gfCNCPoint1[25204] = {X 212.6141, Y 102.4000, Z -2.1667, A 0.000, B 0.000, C 0.000 }
gfCNCPoint1[25205] = {X 194.9870, Y 102.4000, Z -2.1667, A 0.000, B 0.000, C 0.000 }
gfCNCPoint1[25206] = {X 194.0079, Y 102.2897, Z -2.1667, A 0.000, B 0.000, C 0.000 }
gfCNCPoint1[25207] = {X 193.0779, Y 101.9643, Z -2.1667, A 0.000, B 0.000, C 0.000 }
gfCNCPoint1[25208] = {X 192.2436, Y 101.4401, Z -2.1667, A 0.000, B 0.000, C 0.000 }
gfCNCPoint1[25209] = {X 191.5469, Y 100.7434, Z -2.1667, A 0.000, B 0.000, C 0.000 }
gfCNCPoint1[25210] = {X 191.0227, Y 99.9091, Z -2.1667, A 0.000, B 0.000, C 0.000 }
gfCNCPoint1[25211] = {X 190.6973, Y 98.9791, Z -2.1667, A 0.000, B 0.000, C 0.000 }
gfCNCPoint1[25212] = {X 190.5870, Y 98.0000, Z -2.1667, A 0.000, B 0.000, C 0.000 }
gfCNCPoint1[25213] = {X 190.5870, Y 97.0659, Z -2.1667, A 0.000, B 0.000, C 0.000 }
gfCNCPoint1[25214] = {X 190.6897, Y 96.1207, Z -2.1667, A 0.000, B 0.000, C 0.000 }
gfCNCPoint1[25215] = {X 190.9931, Y 95.2196, Z -2.1667, A 0.000, B 0.000, C 0.000 }
gfCNCPoint1[25216] = {X 191.4830, Y 94.4047, Z -2.1667, A 0.000, B 0.000, C 0.000 }
gfCNCPoint1[25217] = {X 188.5295, Y 91.1802, Z -2.1667, A 0.000, B 0.000, C 0.000 }
gfCNCPoint1[25218] = {X 150.1254, Y 91.1802, Z -2.1667, A 0.000, B 0.000, C 0.000 }
gfCNCPoint1[25219] = {X 147.2491, Y 94.3668, Z -2.1667, A 0.000, B 0.000, C 0.000 }
gfCNCPoint1[25220] = {X 147.7550, Y 95.1910, Z -2.1667, A 0.000, B 0.000, C 0.000 }
gfCNCPoint1[25221] = {X 148.0700, Y 96.1053, Z -2.1667, A 0.000, B 0.000, C 0.000 }
gfCNCPoint1[25222] = {X 148.1791, Y 97.0661, Z -2.1667, A 0.000, B 0.000, C 0.000 }
gfCNCPoint1[25223] = {X 148.1791, Y 98.0000, Z -2.1667, A 0.000, B 0.000, C 0.000 }
gfCNCPoint1[25224] = {X 148.0688, Y 98.9791, Z -2.1667, A 0.000, B 0.000, C 0.000 }
gfCNCPoint1[25225] = {X 147.7434, Y 99.9091, Z -2.1667, A 0.000, B 0.000, C 0.000 }
gfCNCPoint1[25226] = {X 147.2192, Y 100.7434, Z -2.1667, A 0.000, B 0.000, C 0.000 }
gfCNCPoint1[25227] = {X 146.5225, Y 101.4401, Z -2.1667, A 0.000, B 0.000, C 0.000 }
gfCNCPoint1[25228] = {X 145.6882, Y 101.9643, Z -2.1667, A 0.000, B 0.000, C 0.000 }
gfCNCPoint1[25229] = {X 144.7582, Y 102.2897, Z -2.1667, A 0.000, B 0.000, C 0.000 }
gfCNCPoint1[25230] = {X 143.7791, Y 102.4000, Z -2.1667, A 0.000, B 0.000, C 0.000 }
gfCNCPoint1[25231] = {X 125.0000, Y 102.4000, Z -2.1667, A 0.000, B 0.000, C 0.000 }
gfCNCPoint1[25232] = {X 124.0209, Y 102.2897, Z -2.1667, A 0.000, B 0.000, C 0.000 }
gfCNCPoint1[25233] = {X 123.0909, Y 101.9643, Z -2.1667, A 0.000, B 0.000, C 0.000 }
gfCNCPoint1[25234] = {X 122.2566, Y 101.4401, Z -2.1667, A 0.000, B 0.000, C 0.000 }
gfCNCPoint1[25235] = {X 121.5599, Y 100.7434, Z -2.1667, A 0.000, B 0.000, C 0.000 }
gfCNCPoint1[25236] = {X 121.0357, Y 99.9091, Z -2.1667, A 0.000, B 0.000, C 0.000 }
gfCNCPoint1[25237] = {X 120.7103, Y 98.9791, Z -2.1667, A 0.000, B 0.000, C 0.000 }
gfCNCPoint1[25238] = {X 120.6000, Y 98.0000, Z -2.1667, A 0.000, B 0.000, C 0.000 }
gfCNCPoint1[25239] = {X 120.6000, Y 97.0659, Z -2.1667, A 0.000, B 0.000, C 0.000 }
gfCNCPoint1[25240] = {X 120.7047, Y 96.1117, Z -2.1667, A 0.000, B 0.000, C 0.000 }
gfCNCPoint1[25241] = {X 121.0139, Y 95.2029, Z -2.1667, A 0.000, B 0.000, C 0.000 }
gfCNCPoint1[25242] = {X 121.5128, Y 94.3828, Z -2.1667, A 0.000, B 0.000, C 0.000 }
gfCNCPoint1[25243] = {X 122.1777, Y 93.6904, Z -2.1667, A 0.000, B 0.000, C 0.000 }
gfCNCPoint1[25244] = {X 122.9769, Y 93.1586, Z -2.1667, A 0.000, B 0.000, C 0.000 }
gfCNCPoint1[25245] = {X 123.8724, Y 92.8129, Z -2.1667, A 0.000, B 0.000, C 0.000 }
gfCNCPoint1[25246] = {X 124.8216, Y 92.6696, Z -2.1667, A 0.000, B 0.000, C 0.000 }
gfCNCPoint1[25247] = {X 124.8681, Y 92.6535, Z -2.1667, A 0.000, B 0.000, C 0.000 }
gfCNCPoint1[25248] = {X 124.9163, Y 92.6433, Z -2.1667, A 0.000, B 0.000, C 0.000 }
gfCNCPoint1[25249] = {X 125.4404, Y 92.5656, Z -2.1667, A 0.000, B 0.000, C 0.000 }
gfCNCPoint1[25250] = {X 126.2564, Y 92.4277, Z -2.1667, A 0.000, B 0.000, C 0.000 }
gfCNCPoint1[25251] = {X 127.0615, Y 92.2363, Z -2.1667, A 0.000, B 0.000, C 0.000 }
gfCNCPoint1[25252] = {X 128.2733, Y 91.0927, Z -2.1667, A 0.000, B 0.000, C 0.000 }
gfCNCPoint1[25253] = {X 129.4217, Y 89.8854, Z -2.1667, A 0.000, B 0.000, C 0.000 }
gfCNCPoint1[25254] = {X 133.5081, Y 85.3901, Z -2.1667, A 0.000, B 0.000, C 0.000 }
gfCNCPoint1[25255] = {X 155.5332, Y 61.2114, Z -2.1667, A 0.000, B 0.000, C 0.000 }
gfCNCPoint1[25256] = {X 155.1842, Y 60.4951, Z -2.1667, A 0.000, B 0.000, C 0.000 }
gfCNCPoint1[25257] = {X 154.9701, Y 59.7276, Z -2.1667, A 0.000, B 0.000, C 0.000 }
gfCNCPoint1[25258] = {X 154.8980, Y 58.9340, Z -2.1667, A 0.000, B 0.000, C 0.000 }
gfCNCPoint1[25259] = {X 154.8980, Y 58.0000, Z -2.1667, A 0.000, B 0.000, C 0.000 }
gfCNCPoint1[25260] = {X 155.0083, Y 57.0209, Z -2.1667, A 0.000, B 0.000, C 0.000 }
gfCNCPoint1[25261] = {X 155.3337, Y 56.0909, Z -2.1667, A 0.000, B 0.000, C 0.000 }
gfCNCPoint1[25262] = {X 155.8579, Y 55.2566, Z -2.1667, A 0.000, B 0.000, C 0.000 }
gfCNCPoint1[25263] = {X 156.5546, Y 54.5599, Z -2.1667, A 0.000, B 0.000, C 0.000 }
gfCNCPoint1[25264] = {X 157.3889, Y 54.0357, Z -2.1667, A 0.000, B 0.000, C 0.000 }
gfCNCPoint1[25265] = {X 158.3189, Y 53.7103, Z -2.1667, A 0.000, B 0.000, C 0.000 }
gfCNCPoint1[25266] = {X 159.2980, Y 53.6000, Z -2.1667, A 0.000, B 0.000, C 0.000 }
gfCNCPoint1[25267] = {X 178.5335, Y 53.6000, Z -2.1667, A 0.000, B 0.000, C 0.000 }
gfCNCPoint1[25268] = {X 179.5126, Y 53.7103, Z -2.1667, A 0.000, B 0.000, C 0.000 }
gfCNCPoint1[25269] = {X 180.4426, Y 54.0357, Z -2.1667, A 0.000, B 0.000, C 0.000 }
gfCNCPoint1[25270] = {X 181.2769, Y 54.5599, Z -2.1667, A 0.000, B 0.000, C 0.000 }
gfCNCPoint1[25271] = {X 181.9736, Y 55.2566, Z -2.1667, A 0.000, B 0.000, C 0.000 }
gfCNCPoint1[25272] = {X 182.4978, Y 56.0909, Z -2.1667, A 0.000, B 0.000, C 0.000 }
gfCNCPoint1[25273] = {X 182.8232, Y 57.0209, Z -2.1667, A 0.000, B 0.000, C 0.000 }
gfCNCPoint1[25274] = {X 182.9335, Y 58.0000, Z -2.1667, A 0.000, B 0.000, C 0.000 }
gfCNCPoint1[25275] = {X 182.9334, Y 58.9704, Z -2.1667, A 0.000, B 0.000, C 0.000 }
gfCNCPoint1[25276] = {X 182.8587, Y 59.7421, Z -2.1667, A 0.000, B 0.000, C 0.000 }
gfCNCPoint1[25277] = {X 182.6497, Y 60.4886, Z -2.1667, A 0.000, B 0.000, C 0.000 }
gfCNCPoint1[25278] = {X 182.3130, Y 61.1869, Z -2.1667, A 0.000, B 0.000, C 0.000 }
gfCNCPoint1[25279] = {X 209.5365, Y 90.8998, Z -2.1667, A 0.000, B 0.000, C 0.000 }
gfCNCPoint1[25280] = {X 210.1906, Y 91.5634, Z -2.1667, A 0.000, B 0.000, C 0.000 }
gfCNCPoint1[25281] = {X 210.8912, Y 92.1776, Z -2.1667, A 0.000, B 0.000, C 0.000 }
gfCNCPoint1[25282] = {X 211.1525, Y 92.3423, Z -2.1667, A 0.000, B 0.000, C 0.000 }
gfCNCPoint1[25283] = {X 211.4457, Y 92.4397, Z -2.1667, A 0.000, B 0.000, C 0.000 }
gfCNCPoint1[25284] = {X 212.1215, Y 92.5841, Z -2.1667, A 0.000, B 0.000, C 0.000 }
gfCNCPoint1[25285] = {X 213.4014, Y 92.7454, Z -2.1667, A 0.000, B 0.000, C 0.000 }
gfCNCPoint1[25286] = {X 214.4545, Y 92.6566, Z -2.1667, A 0.000, B 0.000, C 0.000 }
gfCNCPoint1[25287] = {X 215.5097, Y 92.5965, Z -2.1667, A 0.000, B 0.000, C 0.000 }
gfCNCPoint1[25288] = {X 216.1638, Y 92.5242, Z -2.1667, A 0.000, B 0.000, C 0.000 }
gfCNCPoint1[25289] = {X 216.7936, Y 92.3335, Z -2.1667, A 0.000, B 0.000, C 0.000 }
gfCNCPoint1[25290] = {X 217.3779, Y 92.0307, Z -2.1667, A 0.000, B 0.000, C 0.000 }
gfCNCPoint1[25291] = {X 222.9188, Y 88.4548, Z -2.1667, A 0.000, B 0.000, C 0.000 }
gfCNCPoint1[25292] = {X 245.6538, Y 73.9166, Z -2.1667, A 0.000, B 0.000, C 0.000 }
gfCNCPoint1[25293] = {X 221.6008, Y 64.4770, Z -2.1667, A 0.000, B 0.000, C 0.000 }
gfCNCPoint1[25294] = {X 219.8423, Y 63.8884, Z -2.1667, A 0.000, B 0.000, C 0.000 }
gfCNCPoint1[25295] = {X 218.0280, Y 63.5049, Z -2.1667, A 0.000, B 0.000, C 0.000 }
gfCNCPoint1[25296] = {X 216.1817, Y 63.3315, Z -2.1667, A 0.000, B 0.000, C 0.000 }
gfCNCPoint1[25297] = {X 215.2275, Y 63.1935, Z -2.1667, A 0.000, B 0.000, C 0.000 }
gfCNCPoint1[25298] = {X 214.3263, Y 62.8509, Z -2.1667, A 0.000, B 0.000, C 0.000 }
gfCNCPoint1[25299] = {X 213.5213, Y 62.3203, Z -2.1667, A 0.000, B 0.000, C 0.000 }
gfCNCPoint1[25300] = {X 212.8512, Y 61.6271, Z -2.1667, A 0.000, B 0.000, C 0.000 }
gfCNCPoint1[25301] = {X 212.3482, Y 60.8047, Z -2.1667, A 0.000, B 0.000, C 0.000 }
gfCNCPoint1[25302] = {X 212.0364, Y 59.8924, Z -2.1667, A 0.000, B 0.000, C 0.000 }
gfCNCPoint1[25303] = {X 211.9308, Y 58.9340, Z -2.1667, A 0.000, B 0.000, C 0.000 }
gfCNCPoint1[25304] = {X 211.9308, Y 58.0000, Z -2.1667, A 0.000, B 0.000, C 0.000 }
gfCNCPoint1[25305] = {X 212.0411, Y 57.0209, Z -2.1667, A 0.000, B 0.000, C 0.000 }
gfCNCPoint1[25306] = {X 212.3665, Y 56.0909, Z -2.1667, A 0.000, B 0.000, C 0.000 }
gfCNCPoint1[25307] = {X 212.8907, Y 55.2566, Z -2.1667, A 0.000, B 0.000, C 0.000 }
gfCNCPoint1[25308] = {X 213.5875, Y 54.5599, Z -2.1667, A 0.000, B 0.000, C 0.000 }
gfCNCPoint1[25309] = {X 214.4217, Y 54.0357, Z -2.1667, A 0.000, B 0.000, C 0.000 }
gfCNCPoint1[25310] = {X 215.3517, Y 53.7103, Z -2.1667, A 0.000, B 0.000, C 0.000 }
gfCNCPoint1[25311] = {X 216.3308, Y 53.6000, Z -2.1667, A 0.000, B 0.000, C 0.000 }
gfCNCPoint1[25312] = {X 237.2617, Y 53.6000, Z -2.1667, A 0.000, B 0.000, C 0.000 }
gfCNCPoint1[25313] = {X 238.2408, Y 53.7103, Z -2.1667, A 0.000, B 0.000, C 0.000 }
gfCNCPoint1[25314] = {X 239.1708, Y 54.0357, Z -2.1667, A 0.000, B 0.000, C 0.000 }
gfCNCPoint1[25315] = {X 240.0050, Y 54.5599, Z -2.1667, A 0.000, B 0.000, C 0.000 }
gfCNCPoint1[25316] = {X 240.7017, Y 55.2566, Z -2.1667, A 0.000, B 0.000, C 0.000 }
gfCNCPoint1[25317] = {X 241.2260, Y 56.0909, Z -2.1667, A 0.000, B 0.000, C 0.000 }
gfCNCPoint1[25318] = {X 241.5514, Y 57.0209, Z -2.1667, A 0.000, B 0.000, C 0.000 }
gfCNCPoint1[25319] = {X 241.6617, Y 58.0000, Z -2.1667, A 0.000, B 0.000, C 0.000 }
gfCNCPoint1[25320] = {X 241.6617, Y 58.1782, Z -2.1667, A 0.000, B 0.000, C 0.000 }
gfCNCPoint1[25321] = {X 247.5187, Y 60.4616, Z -2.1667, A 0.000, B 0.000, C 0.000 }
gfCNCPoint1[25322] = {X 275.5538, Y 71.5851, Z -2.1667, A 0.000, B 0.000, C 0.000 }
gfCNCPoint1[25323] = {X 275.5530, Y 63.2813, Z -2.1667, A 0.000, B 0.000, C 0.000 }
gfCNCPoint1[25324] = {X 274.6937, Y 63.0561, Z -2.1667, A 0.000, B 0.000, C 0.000 }
gfCNCPoint1[25325] = {X 273.8971, Y 62.6630, Z -2.1667, A 0.000, B 0.000, C 0.000 }
gfCNCPoint1[25326] = {X 273.1956, Y 62.1178, Z -2.1667, A 0.000, B 0.000, C 0.000 }
gfCNCPoint1[25327] = {X 272.6180, Y 61.4429, Z -2.1667, A 0.000, B 0.000, C 0.000 }
gfCNCPoint1[25328] = {X 272.1877, Y 60.6657, Z -2.1667, A 0.000, B 0.000, C 0.000 }
gfCNCPoint1[25329] = {X 271.9224, Y 59.8179, Z -2.1667, A 0.000, B 0.000, C 0.000 }
gfCNCPoint1[25330] = {X 271.8327, Y 58.9340, Z -2.1667, A 0.000, B 0.000, C 0.000 }
gfCNCPoint1[25331] = {X 271.8327, Y 58.0000, Z -2.1667, A 0.000, B 0.000, C 0.000 }
gfCNCPoint1[25332] = {X 271.9430, Y 57.0209, Z -2.1667, A 0.000, B 0.000, C 0.000 }
gfCNCPoint1[25333] = {X 272.2684, Y 56.0909, Z -2.1667, A 0.000, B 0.000, C 0.000 }
gfCNCPoint1[25334] = {X 272.7926, Y 55.2566, Z -2.1667, A 0.000, B 0.000, C 0.000 }
gfCNCPoint1[25335] = {X 273.4893, Y 54.5599, Z -2.1667, A 0.000, B 0.000, C 0.000 }
gfCNCPoint1[25336] = {X 274.3236, Y 54.0357, Z -2.1667, A 0.000, B 0.000, C 0.000 }
gfCNCPoint1[25337] = {X 275.2536, Y 53.7103, Z -2.1667, A 0.000, B 0.000, C 0.000 }
gfCNCPoint1[25338] = {X 276.2327, Y 53.6000, Z -2.1667, A 0.000, B 0.000, C 0.000 }
gfCNCPoint1[25339] = {X 292.7731, Y 53.6000, Z -2.1667, A 0.000, B 0.000, C 0.000 }
gfCNCPoint1[25340] = {X 293.7522, Y 53.7103, Z -2.1667, A 0.000, B 0.000, C 0.000 }
gfCNCPoint1[25341] = {X 294.6822, Y 54.0357, Z -2.1667, A 0.000, B 0.000, C 0.000 }
gfCNCPoint1[25342] = {X 295.5164, Y 54.5599, Z -2.1667, A 0.000, B 0.000, C 0.000 }
gfCNCPoint1[25343] = {X 296.2131, Y 55.2566, Z -2.1667, A 0.000, B 0.000, C 0.000 }
gfCNCPoint1[25344] = {X 296.7373, Y 56.0909, Z -2.1667, A 0.000, B 0.000, C 0.000 }
gfCNCPoint1[25345] = {X 297.0628, Y 57.0209, Z -2.1667, A 0.000, B 0.000, C 0.000 }
gfCNCPoint1[25346] = {X 297.1731, Y 58.0000, Z -2.1667, A 0.000, B 0.000, C 0.000 }
gfCNCPoint1[25347] = {X 297.1731, Y 58.9355, Z -2.1667, A 0.000, B 0.000, C 0.000 }
gfCNCPoint1[25348] = {X 297.0808, Y 59.8184, Z -2.1667, A 0.000, B 0.000, C 0.000 }
gfCNCPoint1[25349] = {X 296.8139, Y 60.6650, Z -2.1667, A 0.000, B 0.000, C 0.000 }
gfCNCPoint1[25350] = {X 296.3831, Y 61.4411, Z -2.1667, A 0.000, B 0.000, C 0.000 }
gfCNCPoint1[25351] = {X 295.8058, Y 62.1154, Z -2.1667, A 0.000, B 0.000, C 0.000 }
gfCNCPoint1[25352] = {X 295.1053, Y 62.6607, Z -2.1667, A 0.000, B 0.000, C 0.000 }
gfCNCPoint1[25353] = {X 294.3099, Y 63.0548, Z -2.1667, A 0.000, B 0.000, C 0.000 }
gfCNCPoint1[25354] = {X 293.4518, Y 63.2820, Z -2.1667, A 0.000, B 0.000, C 0.000 }
gfCNCPoint1[25355] = {X 293.4518, Y 92.7117, Z -2.1667, A 0.000, B 0.000, C 0.000 }
gfCNCPoint1[25356] = {X 294.3097, Y 92.9414, Z -2.1667, A 0.000, B 0.000, C 0.000 }
gfCNCPoint1[25357] = {X 295.1047, Y 93.3375, Z -2.1667, A 0.000, B 0.000, C 0.000 }
gfCNCPoint1[25358] = {X 295.8047, Y 93.8841, Z -2.1667, A 0.000, B 0.000, C 0.000 }
gfCNCPoint1[25359] = {X 296.3817, Y 94.5592, Z -2.1667, A 0.000, B 0.000, C 0.000 }
gfCNCPoint1[25360] = {X 296.8125, Y 95.3359, Z -2.1667, A 0.000, B 0.000, C 0.000 }
gfCNCPoint1[25361] = {X 297.0799, Y 96.1829, Z -2.1667, A 0.000, B 0.000, C 0.000 }
gfCNCPoint1[25362] = {X 297.1731, Y 97.0661, Z -2.1667, A 0.000, B 0.000, C 0.000 }
gfCNCPoint1[25363] = {X 297.1731, Y 97.6949, Z -2.1667, A 0.000, B 0.000, C 0.000 }
gfCNCPoint1[25364] = {X 297.6531, Y 97.6949, Z -2.1667, A 0.000, B 0.000, C 0.000 }
gfCNCPoint1[25365] = {X 314.2154, Y 97.6949, Z -2.1667, A 0.000, B 0.000, C 0.000 }
gfCNCPoint1[25366] = {X 313.0165, Y 96.8440, Z -2.1667, A 0.000, B 0.000, C 0.000 }
gfCNCPoint1[25367] = {X 311.8816, Y 95.9095, Z -2.1667, A 0.000, B 0.000, C 0.000 }
gfCNCPoint1[25368] = {X 310.9061, Y 94.9480, Z -2.1667, A 0.000, B 0.000, C 0.000 }
gfCNCPoint1[25369] = {X 310.0419, Y 93.8853, Z -2.1667, A 0.000, B 0.000, C 0.000 }
gfCNCPoint1[25370] = {X 309.2079, Y 92.5707, Z -2.1667, A 0.000, B 0.000, C 0.000 }
gfCNCPoint1[25371] = {X 308.5443, Y 91.1624, Z -2.1667, A 0.000, B 0.000, C 0.000 }
gfCNCPoint1[25372] = {X 308.0614, Y 89.6823, Z -2.1667, A 0.000, B 0.000, C 0.000 }
gfCNCPoint1[25373] = {X 307.7080, Y 88.0124, Z -2.1667, A 0.000, B 0.000, C 0.000 }
gfCNCPoint1[25374] = {X 307.4991, Y 86.3184, Z -2.1667, A 0.000, B 0.000, C 0.000 }
gfCNCPoint1[25375] = {X 307.4364, Y 84.6126, Z -2.1667, A 0.000, B 0.000, C 0.000 }
gfCNCPoint1[25376] = {X 307.4376, Y 83.2305, Z -2.1667, A 0.000, B 0.000, C 0.000 }
gfCNCPoint1[25377] = {X 307.4376, Y 63.6745, Z -2.1667, A 0.000, B 0.000, C 0.000 }
gfCNCPoint1[25378] = {X 306.4290, Y 63.3064, Z -2.1667, A 0.000, B 0.000, C 0.000 }
gfCNCPoint1[25379] = {X 305.5253, Y 62.7266, Z -2.1667, A 0.000, B 0.000, C 0.000 }
gfCNCPoint1[25380] = {X 304.7702, Y 61.9632, Z -2.1667, A 0.000, B 0.000, C 0.000 }
gfCNCPoint1[25381] = {X 304.2004, Y 61.0532, Z -2.1667, A 0.000, B 0.000, C 0.000 }
gfCNCPoint1[25382] = {X 303.8433, Y 60.0406, Z -2.1667, A 0.000, B 0.000, C 0.000 }
gfCNCPoint1[25383] = {X 303.7164, Y 58.9744, Z -2.1667, A 0.000, B 0.000, C 0.000 }
gfCNCPoint1[25384] = {X 303.7162, Y 58.0000, Z -2.1667, A 0.000, B 0.000, C 0.000 }
gfCNCPoint1[25385] = {X 303.8100, Y 57.0480, Z -2.1667, A 0.000, B 0.000, C 0.000 }
gfCNCPoint1[25386] = {X 304.0877, Y 56.1325, Z -2.1667, A 0.000, B 0.000, C 0.000 }
gfCNCPoint1[25387] = {X 304.5387, Y 55.2888, Z -2.1667, A 0.000, B 0.000, C 0.000 }
gfCNCPoint1[25388] = {X 305.1455, Y 54.5493, Z -2.1667, A 0.000, B 0.000, C 0.000 }
gfCNCPoint1[25389] = {X 305.8850, Y 53.9424, Z -2.1667, A 0.000, B 0.000, C 0.000 }
gfCNCPoint1[25390] = {X 306.7287, Y 53.4915, Z -2.1667, A 0.000, B 0.000, C 0.000 }
gfCNCPoint1[25391] = {X 307.6442, Y 53.2138, Z -2.1667, A 0.000, B 0.000, C 0.000 }
gfCNCPoint1[25392] = {X 308.5962, Y 53.1200, Z -2.1667, A 0.000, B 0.000, C 0.000 }
gfCNCPoint1[25393] = {X 324.3107, Y 53.1200, Z -2.1667, A 0.000, B 0.000, C 0.000 }
gfCNCPoint1[25394] = {X 325.2627, Y 53.2138, Z -2.1667, A 0.000, B 0.000, C 0.000 }
gfCNCPoint1[25395] = {X 326.1782, Y 53.4915, Z -2.1667, A 0.000, B 0.000, C 0.000 }
gfCNCPoint1[25396] = {X 327.0219, Y 53.9424, Z -2.1667, A 0.000, B 0.000, C 0.000 }
gfCNCPoint1[25397] = {X 327.7614, Y 54.5493, Z -2.1667, A 0.000, B 0.000, C 0.000 }
gfCNCPoint1[25398] = {X 328.3683, Y 55.2888, Z -2.1667, A 0.000, B 0.000, C 0.000 }
gfCNCPoint1[25399] = {X 328.8192, Y 56.1325, Z -2.1667, A 0.000, B 0.000, C 0.000 }
gfCNCPoint1[25400] = {X 329.0969, Y 57.0480, Z -2.1667, A 0.000, B 0.000, C 0.000 }
gfCNCPoint1[25401] = {X 329.1907, Y 58.0000, Z -2.1667, A 0.000, B 0.000, C 0.000 }
gfCNCPoint1[25402] = {X 329.1907, Y 58.9341, Z -2.1667, A 0.000, B 0.000, C 0.000 }
gfCNCPoint1[25403] = {X 329.0668, Y 60.0066, Z -2.1667, A 0.000, B 0.000, C 0.000 }
gfCNCPoint1[25404] = {X 328.7119, Y 61.0263, Z -2.1667, A 0.000, B 0.000, C 0.000 }
gfCNCPoint1[25405] = {X 328.1432, Y 61.9440, Z -2.1667, A 0.000, B 0.000, C 0.000 }
gfCNCPoint1[25406] = {X 327.3880, Y 62.7155, Z -2.1667, A 0.000, B 0.000, C 0.000 }
gfCNCPoint1[25407] = {X 326.4827, Y 63.3037, Z -2.1667, A 0.000, B 0.000, C 0.000 }
gfCNCPoint1[25408] = {X 325.4708, Y 63.6803, Z -2.1667, A 0.000, B 0.000, C 0.000 }
gfCNCPoint1[25409] = {X 325.4722, Y 83.2268, Z -2.1667, A 0.000, B 0.000, C 0.000 }
gfCNCPoint1[25410] = {X 325.4857, Y 84.6073, Z -2.1667, A 0.000, B 0.000, C 0.000 }
gfCNCPoint1[25411] = {X 325.5516, Y 85.7202, Z -2.1667, A 0.000, B 0.000, C 0.000 }
gfCNCPoint1[25412] = {X 325.7423, Y 86.8186, Z -2.1667, A 0.000, B 0.000, C 0.000 }
gfCNCPoint1[25413] = {X 325.8862, Y 86.9530, Z -2.1667, A 0.000, B 0.000, C 0.000 }
gfCNCPoint1[25414] = {X 326.0544, Y 87.0553, Z -2.1667, A 0.000, B 0.000, C 0.000 }
gfCNCPoint1[25415] = {X 326.4828, Y 87.2970, Z -2.1667, A 0.000, B 0.000, C 0.000 }
gfCNCPoint1[25416] = {X 327.8562, Y 87.8661, Z -2.1667, A 0.000, B 0.000, C 0.000 }
gfCNCPoint1[25417] = {X 329.2836, Y 88.2815, Z -2.1667, A 0.000, B 0.000, C 0.000 }
gfCNCPoint1[25418] = {X 332.3214, Y 88.8899, Z -2.1667, A 0.000, B 0.000, C 0.000 }
gfCNCPoint1[25419] = {X 335.3952, Y 89.2776, Z -2.1667, A 0.000, B 0.000, C 0.000 }
gfCNCPoint1[25420] = {X 339.5150, Y 89.5954, Z -2.1667, A 0.000, B 0.000, C 0.000 }
gfCNCPoint1[25421] = {X 343.6432, Y 89.7744, Z -2.1667, A 0.000, B 0.000, C 0.000 }
gfCNCPoint1[25422] = {X 347.7751, Y 89.8144, Z -2.1667, A 0.000, B 0.000, C 0.000 }
gfCNCPoint1[25423] = {X 352.1401, Y 89.7764, Z -2.1667, A 0.000, B 0.000, C 0.000 }
gfCNCPoint1[25424] = {X 356.5009, Y 89.5815, Z -2.1667, A 0.000, B 0.000, C 0.000 }
gfCNCPoint1[25425] = {X 360.8519, Y 89.2298, Z -2.1667, A 0.000, B 0.000, C 0.000 }
gfCNCPoint1[25426] = {X 363.1336, Y 88.9461, Z -2.1667, A 0.000, B 0.000, C 0.000 }
gfCNCPoint1[25427] = {X 365.3941, Y 88.5258, Z -2.1667, A 0.000, B 0.000, C 0.000 }
gfCNCPoint1[25428] = {X 367.6252, Y 87.9704, Z -2.1667, A 0.000, B 0.000, C 0.000 }
gfCNCPoint1[25429] = {X 368.9191, Y 87.4953, Z -2.1667, A 0.000, B 0.000, C 0.000 }
gfCNCPoint1[25430] = {X 370.1149, Y 86.8101, Z -2.1667, A 0.000, B 0.000, C 0.000 }
gfCNCPoint1[25431] = {X 370.2995, Y 85.3240, Z -2.1667, A 0.000, B 0.000, C 0.000 }
gfCNCPoint1[25432] = {X 370.3611, Y 83.8278, Z -2.1667, A 0.000, B 0.000, C 0.000 }
gfCNCPoint1[25433] = {X 370.3594, Y 63.6742, Z -2.1667, A 0.000, B 0.000, C 0.000 }
gfCNCPoint1[25434] = {X 369.3511, Y 63.3059, Z -2.1667, A 0.000, B 0.000, C 0.000 }
gfCNCPoint1[25435] = {X 368.4476, Y 62.7261, Z -2.1667, A 0.000, B 0.000, C 0.000 }
gfCNCPoint1[25436] = {X 367.6928, Y 61.9627, Z -2.1667, A 0.000, B 0.000, C 0.000 }
gfCNCPoint1[25437] = {X 367.1232, Y 61.0528, Z -2.1667, A 0.000, B 0.000, C 0.000 }
gfCNCPoint1[25438] = {X 366.7663, Y 60.0404, Z -2.1667, A 0.000, B 0.000, C 0.000 }
gfCNCPoint1[25439] = {X 366.6394, Y 58.9744, Z -2.1667, A 0.000, B 0.000, C 0.000 }
gfCNCPoint1[25440] = {X 366.6393, Y 58.0000, Z -2.1667, A 0.000, B 0.000, C 0.000 }
gfCNCPoint1[25441] = {X 366.7331, Y 57.0480, Z -2.1667, A 0.000, B 0.000, C 0.000 }
gfCNCPoint1[25442] = {X 367.0108, Y 56.1325, Z -2.1667, A 0.000, B 0.000, C 0.000 }
gfCNCPoint1[25443] = {X 367.4617, Y 55.2888, Z -2.1667, A 0.000, B 0.000, C 0.000 }
gfCNCPoint1[25444] = {X 368.0686, Y 54.5493, Z -2.1667, A 0.000, B 0.000, C 0.000 }
gfCNCPoint1[25445] = {X 368.8081, Y 53.9424, Z -2.1667, A 0.000, B 0.000, C 0.000 }
gfCNCPoint1[25446] = {X 369.6518, Y 53.4915, Z -2.1667, A 0.000, B 0.000, C 0.000 }
gfCNCPoint1[25447] = {X 370.5672, Y 53.2138, Z -2.1667, A 0.000, B 0.000, C 0.000 }
gfCNCPoint1[25448] = {X 371.5193, Y 53.1200, Z -2.1667, A 0.000, B 0.000, C 0.000 }
gfCNCPoint1[25449] = {X 388.0597, Y 53.1200, Z -2.1667, A 0.000, B 0.000, C 0.000 }
gfCNCPoint1[25450] = {X 389.0355, Y 53.2186, Z -2.1667, A 0.000, B 0.000, C 0.000 }
gfCNCPoint1[25451] = {X 389.9719, Y 53.5102, Z -2.1667, A 0.000, B 0.000, C 0.000 }
gfCNCPoint1[25452] = {X 390.8310, Y 53.9833, Z -2.1667, A 0.000, B 0.000, C 0.000 }
gfCNCPoint1[25453] = {X 391.5783, Y 54.6186, Z -2.1667, A 0.000, B 0.000, C 0.000 }
gfCNCPoint1[25454] = {X 392.1572, Y 55.3496, Z -2.1667, A 0.000, B 0.000, C 0.000 }
gfCNCPoint1[25455] = {X 392.5865, Y 56.1774, Z -2.1667, A 0.000, B 0.000, C 0.000 }
gfCNCPoint1[25456] = {X 392.8506, Y 57.0718, Z -2.1667, A 0.000, B 0.000, C 0.000 }
gfCNCPoint1[25457] = {X 392.9397, Y 58.0000, Z -2.1667, A 0.000, B 0.000, C 0.000 }
gfCNCPoint1[25458] = {X 392.9395, Y 58.9744, Z -2.1667, A 0.000, B 0.000, C 0.000 }
gfCNCPoint1[25459] = {X 392.8773, Y 59.7118, Z -2.1667, A 0.000, B 0.000, C 0.000 }
gfCNCPoint1[25460] = {X 392.7043, Y 60.4314, Z -2.1667, A 0.000, B 0.000, C 0.000 }
gfCNCPoint1[25461] = {X 392.4245, Y 61.1165, Z -2.1667, A 0.000, B 0.000, C 0.000 }
gfCNCPoint1[25462] = {X 392.0463, Y 61.7490, Z -2.1667, A 0.000, B 0.000, C 0.000 }
gfCNCPoint1[25463] = {X 391.5775, Y 62.3176, Z -2.1667, A 0.000, B 0.000, C 0.000 }
gfCNCPoint1[25464] = {X 390.8816, Y 62.9184, Z -2.1667, A 0.000, B 0.000, C 0.000 }
gfCNCPoint1[25465] = {X 390.0858, Y 63.3787, Z -2.1667, A 0.000, B 0.000, C 0.000 }
gfCNCPoint1[25466] = {X 389.2180, Y 63.6822, Z -2.1667, A 0.000, B 0.000, C 0.000 }
gfCNCPoint1[25467] = {X 389.2159, Y 84.6140, Z -2.1667, A 0.000, B 0.000, C 0.000 }
gfCNCPoint1[25468] = {X 389.1537, Y 86.3200, Z -2.1667, A 0.000, B 0.000, C 0.000 }
gfCNCPoint1[25469] = {X 388.9434, Y 88.0140, Z -2.1667, A 0.000, B 0.000, C 0.000 }
gfCNCPoint1[25470] = {X 388.5865, Y 89.6834, Z -2.1667, A 0.000, B 0.000, C 0.000 }
gfCNCPoint1[25471] = {X 388.1034, Y 91.1629, Z -2.1667, A 0.000, B 0.000, C 0.000 }
gfCNCPoint1[25472] = {X 387.4397, Y 92.5708, Z -2.1667, A 0.000, B 0.000, C 0.000 }
gfCNCPoint1[25473] = {X 386.6057, Y 93.8849, Z -2.1667, A 0.000, B 0.000, C 0.000 }
gfCNCPoint1[25474] = {X 385.8732, Y 94.7999, Z -2.1667, A 0.000, B 0.000, C 0.000 }
gfCNCPoint1[25475] = {X 385.0580, Y 95.6421, Z -2.1667, A 0.000, B 0.000, C 0.000 }
gfCNCPoint1[25476] = {X 383.7980, Y 96.7250, Z -2.1667, A 0.000, B 0.000, C 0.000 }
gfCNCPoint1[25477] = {X 382.4492, Y 97.6949, Z -2.1667, A 0.000, B 0.000, C 0.000 }
gfCNCPoint1[25478] = {X 382.1861, Y 97.2934, Z -2.1667, A 0.000, B 0.000, C 0.000 }
gfCNCPoint1[25479] = {X 381.0192, Y 97.9987, Z -2.1667, A 0.000, B 0.000, C 0.000 }
gfCNCPoint1[25480] = {X 379.8040, Y 98.6171, Z -2.1667, A 0.000, B 0.000, C 0.000 }
gfCNCPoint1[25481] = {X 377.5271, Y 99.5757, Z -2.1667, A 0.000, B 0.000, C 0.000 }
gfCNCPoint1[25482] = {X 375.1871, Y 100.3679, Z -2.1667, A 0.000, B 0.000, C 0.000 }
gfCNCPoint1[25483] = {X 372.7962, Y 100.9897, Z -2.1667, A 0.000, B 0.000, C 0.000 }
gfCNCPoint1[25484] = {X 368.9811, Y 101.7277, Z -2.1667, A 0.000, B 0.000, C 0.000 }
gfCNCPoint1[25485] = {X 365.1349, Y 102.2816, Z -2.1667, A 0.000, B 0.000, C 0.000 }
gfCNCPoint1[25486] = {X 361.2665, Y 102.6498, Z -2.1667, A 0.000, B 0.000, C 0.000 }
gfCNCPoint1[25487] = {X 355.1239, Y 102.9832, Z -2.1667, A 0.000, B 0.000, C 0.000 }
gfCNCPoint1[25488] = {X 348.9737, Y 103.1117, Z -2.1667, A 0.000, B 0.000, C 0.000 }
gfCNCPoint1[25489] = {X 342.8225, Y 103.0353, Z -2.1667, A 0.000, B 0.000, C 0.000 }
gfCNCPoint1[25490] = {X 336.6774, Y 102.7540, Z -2.1667, A 0.000, B 0.000, C 0.000 }
gfCNCPoint1[25491] = {X 333.1844, Y 102.4787, Z -2.1667, A 0.000, B 0.000, C 0.000 }
gfCNCPoint1[25492] = {X 329.7050, Y 102.0654, Z -2.1667, A 0.000, B 0.000, C 0.000 }
gfCNCPoint1[25493] = {X 326.2448, Y 101.5147, Z -2.1667, A 0.000, B 0.000, C 0.000 }
gfCNCPoint1[25494] = {X 323.3896, Y 100.9088, Z -2.1667, A 0.000, B 0.000, C 0.000 }
gfCNCPoint1[25495] = {X 320.5868, Y 100.0943, Z -2.1667, A 0.000, B 0.000, C 0.000 }
gfCNCPoint1[25496] = {X 317.8517, Y 99.0755, Z -2.1667, A 0.000, B 0.000, C 0.000 }
gfCNCPoint1[25497] = {X 316.3330, Y 98.3746, Z -2.1667, A 0.000, B 0.000, C 0.000 }
gfCNCPoint1[25498] = {X 314.8782, Y 97.5494, Z -2.1667, A 0.000, B 0.000, C 0.000 }
gfCNCPoint1[25499] = {X 313.4972, Y 96.6057, Z -2.1667, A 0.000, B 0.000, C 0.000 }
gfCNCPoint1[25500] = {X 312.1998, Y 95.5501, Z -2.1667, A 0.000, B 0.000, C 0.000 }
gfCNCPoint1[25501] = {X 311.1892, Y 94.5452, Z -2.1667, A 0.000, B 0.000, C 0.000 }
gfCNCPoint1[25502] = {X 310.3051, Y 93.4274, Z -2.1667, A 0.000, B 0.000, C 0.000 }
gfCNCPoint1[25503] = {X 309.5598, Y 92.2126, Z -2.1667, A 0.000, B 0.000, C 0.000 }
gfCNCPoint1[25504] = {X 308.9640, Y 90.9179, Z -2.1667, A 0.000, B 0.000, C 0.000 }
gfCNCPoint1[25505] = {X 308.5260, Y 89.5616, Z -2.1667, A 0.000, B 0.000, C 0.000 }
gfCNCPoint1[25506] = {X 308.1812, Y 87.9321, Z -2.1667, A 0.000, B 0.000, C 0.000 }
gfCNCPoint1[25507] = {X 307.9775, Y 86.2789, Z -2.1667, A 0.000, B 0.000, C 0.000 }
gfCNCPoint1[25508] = {X 307.9164, Y 84.6144, Z -2.1667, A 0.000, B 0.000, C 0.000 }
gfCNCPoint1[25509] = {X 307.9176, Y 83.2309, Z -2.1667, A 0.000, B 0.000, C 0.000 }
gfCNCPoint1[25510] = {X 307.9176, Y 63.2814, Z -2.1667, A 0.000, B 0.000, C 0.000 }
gfCNCPoint1[25511] = {X 307.0581, Y 63.0565, Z -2.1667, A 0.000, B 0.000, C 0.000 }
gfCNCPoint1[25512] = {X 306.2612, Y 62.6634, Z -2.1667, A 0.000, B 0.000, C 0.000 }
gfCNCPoint1[25513] = {X 305.5596, Y 62.1182, Z -2.1667, A 0.000, B 0.000, C 0.000 }
gfCNCPoint1[25514] = {X 304.9818, Y 61.4433, Z -2.1667, A 0.000, B 0.000, C 0.000 }
gfCNCPoint1[25515] = {X 304.5514, Y 60.6660, Z -2.1667, A 0.000, B 0.000, C 0.000 }
gfCNCPoint1[25516] = {X 304.2859, Y 59.8180, Z -2.1667, A 0.000, B 0.000, C 0.000 }
gfCNCPoint1[25517] = {X 304.1962, Y 58.9340, Z -2.1667, A 0.000, B 0.000, C 0.000 }
gfCNCPoint1[25518] = {X 304.1962, Y 58.0000, Z -2.1667, A 0.000, B 0.000, C 0.000 }
gfCNCPoint1[25519] = {X 304.3065, Y 57.0209, Z -2.1667, A 0.000, B 0.000, C 0.000 }
gfCNCPoint1[25520] = {X 304.6320, Y 56.0909, Z -2.1667, A 0.000, B 0.000, C 0.000 }
gfCNCPoint1[25521] = {X 305.1562, Y 55.2566, Z -2.1667, A 0.000, B 0.000, C 0.000 }
gfCNCPoint1[25522] = {X 305.8529, Y 54.5599, Z -2.1667, A 0.000, B 0.000, C 0.000 }
gfCNCPoint1[25523] = {X 306.6871, Y 54.0357, Z -2.1667, A 0.000, B 0.000, C 0.000 }
gfCNCPoint1[25524] = {X 307.6171, Y 53.7103, Z -2.1667, A 0.000, B 0.000, C 0.000 }
gfCNCPoint1[25525] = {X 308.5962, Y 53.6000, Z -2.1667, A 0.000, B 0.000, C 0.000 }
gfCNCPoint1[25526] = {X 324.3107, Y 53.6000, Z -2.1667, A 0.000, B 0.000, C 0.000 }
gfCNCPoint1[25527] = {X 325.2898, Y 53.7103, Z -2.1667, A 0.000, B 0.000, C 0.000 }
gfCNCPoint1[25528] = {X 326.2198, Y 54.0357, Z -2.1667, A 0.000, B 0.000, C 0.000 }
gfCNCPoint1[25529] = {X 327.0540, Y 54.5599, Z -2.1667, A 0.000, B 0.000, C 0.000 }
gfCNCPoint1[25530] = {X 327.7507, Y 55.2566, Z -2.1667, A 0.000, B 0.000, C 0.000 }
gfCNCPoint1[25531] = {X 328.2750, Y 56.0909, Z -2.1667, A 0.000, B 0.000, C 0.000 }
gfCNCPoint1[25532] = {X 328.6004, Y 57.0209, Z -2.1667, A 0.000, B 0.000, C 0.000 }
gfCNCPoint1[25533] = {X 328.7107, Y 58.0000, Z -2.1667, A 0.000, B 0.000, C 0.000 }
gfCNCPoint1[25534] = {X 328.7107, Y 58.9366, Z -2.1667, A 0.000, B 0.000, C 0.000 }
gfCNCPoint1[25535] = {X 328.6165, Y 59.8191, Z -2.1667, A 0.000, B 0.000, C 0.000 }
gfCNCPoint1[25536] = {X 328.3487, Y 60.6654, Z -2.1667, A 0.000, B 0.000, C 0.000 }
gfCNCPoint1[25537] = {X 327.9178, Y 61.4414, Z -2.1667, A 0.000, B 0.000, C 0.000 }
gfCNCPoint1[25538] = {X 327.3413, Y 62.1162, Z -2.1667, A 0.000, B 0.000, C 0.000 }
gfCNCPoint1[25539] = {X 326.6420, Y 62.6628, Z -2.1667, A 0.000, B 0.000, C 0.000 }
gfCNCPoint1[25540] = {X 325.8479, Y 63.0594, Z -2.1667, A 0.000, B 0.000, C 0.000 }
gfCNCPoint1[25541] = {X 324.9908, Y 63.2901, Z -2.1667, A 0.000, B 0.000, C 0.000 }
gfCNCPoint1[25542] = {X 324.9922, Y 83.2292, Z -2.1667, A 0.000, B 0.000, C 0.000 }
gfCNCPoint1[25543] = {X 325.0058, Y 84.6146, Z -2.1667, A 0.000, B 0.000, C 0.000 }
gfCNCPoint1[25544] = {X 325.0816, Y 85.8327, Z -2.1667, A 0.000, B 0.000, C 0.000 }
gfCNCPoint1[25545] = {X 325.3001, Y 87.0335, Z -2.1667, A 0.000, B 0.000, C 0.000 }
gfCNCPoint1[25546] = {X 325.5330, Y 87.2843, Z -2.1667, A 0.000, B 0.000, C 0.000 }
gfCNCPoint1[25547] = {X 325.8185, Y 87.4733, Z -2.1667, A 0.000, B 0.000, C 0.000 }
gfCNCPoint1[25548] = {X 326.2606, Y 87.7228, Z -2.1667, A 0.000, B 0.000, C 0.000 }
gfCNCPoint1[25549] = {X 327.6904, Y 88.3166, Z -2.1667, A 0.000, B 0.000, C 0.000 }
gfCNCPoint1[25550] = {X 329.1769, Y 88.7495, Z -2.1667, A 0.000, B 0.000, C 0.000 }
gfCNCPoint1[25551] = {X 332.2474, Y 89.3642, Z -2.1667, A 0.000, B 0.000, C 0.000 }
gfCNCPoint1[25552] = {X 335.3541, Y 89.7558, Z -2.1667, A 0.000, B 0.000, C 0.000 }
gfCNCPoint1[25553] = {X 339.4910, Y 90.0748, Z -2.1667, A 0.000, B 0.000, C 0.000 }
gfCNCPoint1[25554] = {X 343.6362, Y 90.2544, Z -2.1667, A 0.000, B 0.000, C 0.000 }
gfCNCPoint1[25555] = {X 347.7851, Y 90.2944, Z -2.1667, A 0.000, B 0.000, C 0.000 }
gfCNCPoint1[25556] = {X 352.1632, Y 90.2559, Z -2.1667, A 0.000, B 0.000, C 0.000 }
gfCNCPoint1[25557] = {X 356.5371, Y 90.0601, Z -2.1667, A 0.000, B 0.000, C 0.000 }
gfCNCPoint1[25558] = {X 360.9012, Y 89.7072, Z -2.1667, A 0.000, B 0.000, C 0.000 }
gfCNCPoint1[25559] = {X 363.2108, Y 89.4199, Z -2.1667, A 0.000, B 0.000, C 0.000 }
gfCNCPoint1[25560] = {X 365.4989, Y 88.9943, Z -2.1667, A 0.000, B 0.000, C 0.000 }
gfCNCPoint1[25561] = {X 367.7574, Y 88.4318, Z -2.1667, A 0.000, B 0.000, C 0.000 }
gfCNCPoint1[25562] = {X 368.6804, Y 88.1214, Z -2.1667, A 0.000, B 0.000, C 0.000 }
gfCNCPoint1[25563] = {X 369.5628, Y 87.7094, Z -2.1667, A 0.000, B 0.000, C 0.000 }
gfCNCPoint1[25564] = {X 370.3934, Y 87.2011, Z -2.1667, A 0.000, B 0.000, C 0.000 }
gfCNCPoint1[25565] = {X 370.5214, Y 87.0679, Z -2.1667, A 0.000, B 0.000, C 0.000 }
gfCNCPoint1[25566] = {X 370.5873, Y 86.8954, Z -2.1667, A 0.000, B 0.000, C 0.000 }
gfCNCPoint1[25567] = {X 370.7776, Y 85.3669, Z -2.1667, A 0.000, B 0.000, C 0.000 }
gfCNCPoint1[25568] = {X 370.8411, Y 83.8278, Z -2.1667, A 0.000, B 0.000, C 0.000 }
gfCNCPoint1[25569] = {X 370.8394, Y 63.2812, Z -2.1667, A 0.000, B 0.000, C 0.000 }
gfCNCPoint1[25570] = {X 369.9801, Y 63.0561, Z -2.1667, A 0.000, B 0.000, C 0.000 }
gfCNCPoint1[25571] = {X 369.1835, Y 62.6629, Z -2.1667, A 0.000, B 0.000, C 0.000 }
gfCNCPoint1[25572] = {X 368.4821, Y 62.1177, Z -2.1667, A 0.000, B 0.000, C 0.000 }
gfCNCPoint1[25573] = {X 367.9046, Y 61.4428, Z -2.1667, A 0.000, B 0.000, C 0.000 }
gfCNCPoint1[25574] = {X 367.4743, Y 60.6656, Z -2.1667, A 0.000, B 0.000, C 0.000 }
gfCNCPoint1[25575] = {X 367.2090, Y 59.8178, Z -2.1667, A 0.000, B 0.000, C 0.000 }
gfCNCPoint1[25576] = {X 367.1193, Y 58.9340, Z -2.1667, A 0.000, B 0.000, C 0.000 }
gfCNCPoint1[25577] = {X 367.1193, Y 58.0000, Z -2.1667, A 0.000, B 0.000, C 0.000 }
gfCNCPoint1[25578] = {X 367.2296, Y 57.0209, Z -2.1667, A 0.000, B 0.000, C 0.000 }
gfCNCPoint1[25579] = {X 367.5550, Y 56.0909, Z -2.1667, A 0.000, B 0.000, C 0.000 }
gfCNCPoint1[25580] = {X 368.0792, Y 55.2566, Z -2.1667, A 0.000, B 0.000, C 0.000 }
gfCNCPoint1[25581] = {X 368.7759, Y 54.5599, Z -2.1667, A 0.000, B 0.000, C 0.000 }
gfCNCPoint1[25582] = {X 369.6102, Y 54.0357, Z -2.1667, A 0.000, B 0.000, C 0.000 }
gfCNCPoint1[25583] = {X 370.5402, Y 53.7103, Z -2.1667, A 0.000, B 0.000, C 0.000 }
gfCNCPoint1[25584] = {X 371.5193, Y 53.6000, Z -2.1667, A 0.000, B 0.000, C 0.000 }
gfCNCPoint1[25585] = {X 388.0597, Y 53.6000, Z -2.1667, A 0.000, B 0.000, C 0.000 }
gfCNCPoint1[25586] = {X 389.0388, Y 53.7103, Z -2.1667, A 0.000, B 0.000, C 0.000 }
gfCNCPoint1[25587] = {X 389.9688, Y 54.0357, Z -2.1667, A 0.000, B 0.000, C 0.000 }
gfCNCPoint1[25588] = {X 390.8030, Y 54.5599, Z -2.1667, A 0.000, B 0.000, C 0.000 }
gfCNCPoint1[25589] = {X 391.4997, Y 55.2566, Z -2.1667, A 0.000, B 0.000, C 0.000 }
gfCNCPoint1[25590] = {X 392.0239, Y 56.0909, Z -2.1667, A 0.000, B 0.000, C 0.000 }
gfCNCPoint1[25591] = {X 392.3494, Y 57.0209, Z -2.1667, A 0.000, B 0.000, C 0.000 }
gfCNCPoint1[25592] = {X 392.4597, Y 58.0000, Z -2.1667, A 0.000, B 0.000, C 0.000 }
gfCNCPoint1[25593] = {X 392.4595, Y 58.9704, Z -2.1667, A 0.000, B 0.000, C 0.000 }
gfCNCPoint1[25594] = {X 392.3378, Y 59.9627, Z -2.1667, A 0.000, B 0.000, C 0.000 }
gfCNCPoint1[25595] = {X 391.9951, Y 60.9018, Z -2.1667, A 0.000, B 0.000, C 0.000 }
gfCNCPoint1[25596] = {X 391.5512, Y 61.6122, Z -2.1667, A 0.000, B 0.000, C 0.000 }
gfCNCPoint1[25597] = {X 390.9813, Y 62.2261, Z -2.1667, A 0.000, B 0.000, C 0.000 }
gfCNCPoint1[25598] = {X 390.3058, Y 62.7215, Z -2.1667, A 0.000, B 0.000, C 0.000 }
gfCNCPoint1[25599] = {X 389.5489, Y 63.0805, Z -2.1667, A 0.000, B 0.000, C 0.000 }
gfCNCPoint1[25600] = {X 388.7380, Y 63.2904, Z -2.1667, A 0.000, B 0.000, C 0.000 }
gfCNCPoint1[25601] = {X 388.7380, Y 83.9247, Z -2.1667, A 0.000, B 0.000, C 0.000 }
gfCNCPoint1[25602] = {X 388.7359, Y 84.6150, Z -2.1667, A 0.000, B 0.000, C 0.000 }
gfCNCPoint1[25603] = {X 388.6754, Y 86.2800, Z -2.1667, A 0.000, B 0.000, C 0.000 }
gfCNCPoint1[25604] = {X 388.4702, Y 87.9334, Z -2.1667, A 0.000, B 0.000, C 0.000 }
gfCNCPoint1[25605] = {X 388.1219, Y 89.5627, Z -2.1667, A 0.000, B 0.000, C 0.000 }
gfCNCPoint1[25606] = {X 387.5862, Y 91.1608, Z -2.1667, A 0.000, B 0.000, C 0.000 }
gfCNCPoint1[25607] = {X 386.8315, Y 92.6680, Z -2.1667, A 0.000, B 0.000, C 0.000 }
gfCNCPoint1[25608] = {X 385.8729, Y 94.0543, Z -2.1667, A 0.000, B 0.000, C 0.000 }
gfCNCPoint1[25609] = {X 384.7292, Y 95.2925, Z -2.1667, A 0.000, B 0.000, C 0.000 }
gfCNCPoint1[25610] = {X 383.5010, Y 96.3480, Z -2.1667, A 0.000, B 0.000, C 0.000 }
gfCNCPoint1[25611] = {X 382.1861, Y 97.2934, Z -2.1667, A 0.000, B 0.000, C 0.000 }
gfCNCPoint1[25612] = {X 382.4492, Y 97.6949, Z -2.1667, A 0.000, B 0.000, C 0.000 }
gfCNCPoint1[25613] = {X 391.5259, Y 97.6949, Z -2.1667, A 0.000, B 0.000, C 0.000 }
gfCNCPoint1[25614] = {X 391.5259, Y 97.0659, Z -2.1667, A 0.000, B 0.000, C 0.000 }
gfCNCPoint1[25615] = {X 391.6192, Y 96.1165, Z -2.1667, A 0.000, B 0.000, C 0.000 }
gfCNCPoint1[25616] = {X 391.8954, Y 95.2034, Z -2.1667, A 0.000, B 0.000, C 0.000 }
gfCNCPoint1[25617] = {X 392.3439, Y 94.3615, Z -2.1667, A 0.000, B 0.000, C 0.000 }
gfCNCPoint1[25618] = {X 392.9477, Y 93.6229, Z -2.1667, A 0.000, B 0.000, C 0.000 }
gfCNCPoint1[25619] = {X 393.6836, Y 93.0158, Z -2.1667, A 0.000, B 0.000, C 0.000 }
gfCNCPoint1[25620] = {X 394.5236, Y 92.5636, Z -2.1667, A 0.000, B 0.000, C 0.000 }
gfCNCPoint1[25621] = {X 395.4355, Y 92.2834, Z -2.1667, A 0.000, B 0.000, C 0.000 }
gfCNCPoint1[25622] = {X 396.3845, Y 92.1860, Z -2.1667, A 0.000, B 0.000, C 0.000 }
gfCNCPoint1[25623] = {X 397.3062, Y 92.1468, Z -2.1667, A 0.000, B 0.000, C 0.000 }
gfCNCPoint1[25624] = {X 398.2245, Y 92.0596, Z -2.1667, A 0.000, B 0.000, C 0.000 }
gfCNCPoint1[25625] = {X 398.7527, Y 91.9314, Z -2.1667, A 0.000, B 0.000, C 0.000 }
gfCNCPoint1[25626] = {X 399.2389, Y 91.6888, Z -2.1667, A 0.000, B 0.000, C 0.000 }
gfCNCPoint1[25627] = {X 426.8279, Y 74.0193, Z -2.1667, A 0.000, B 0.000, C 0.000 }
gfCNCPoint1[25628] = {X 403.5508, Y 64.8861, Z -2.1667, A 0.000, B 0.000, C 0.000 }
gfCNCPoint1[25629] = {X 402.0005, Y 64.3678, Z -2.1667, A 0.000, B 0.000, C 0.000 }
gfCNCPoint1[25630] = {X 400.4046, Y 64.0138, Z -2.1667, A 0.000, B 0.000, C 0.000 }
gfCNCPoint1[25631] = {X 398.8170, Y 73.4816, Z -2.1667, A 0.000, B 0.000, C 0.000 }
gfCNCPoint1[25632] = {X 398.8163, Y 80.5594, Z -2.1667, A 0.000, B 0.000, C 0.000 }
gfCNCPoint1[25633] = {X 405.8053, Y 76.0832, Z -2.1667, A 0.000, B 0.000, C 0.000 }
gfCNCPoint1[25634] = {X 400.0363, Y 73.8196, Z -2.1667, A 0.000, B 0.000, C 0.000 }
gfCNCPoint1[25635] = {X 399.4355, Y 73.6188, Z -2.1667, A 0.000, B 0.000, C 0.000 }
gfCNCPoint1[25636] = {X 398.8170, Y 73.4816, Z -2.1667, A 0.000, B 0.000, C 0.000 }
gfCNCPoint1[25637] = {X 399.2139, Y 71.1146, Z -2.1667, A 0.000, B 0.000, C 0.000 }
gfCNCPoint1[25638] = {X 398.7491, Y 71.0498, Z -2.1667, A 0.000, B 0.000, C 0.000 }
gfCNCPoint1[25639] = {X 398.2813, Y 71.0109, Z -2.1667, A 0.000, B 0.000, C 0.000 }
gfCNCPoint1[25640] = {X 397.3456, Y 70.9531, Z -2.1667, A 0.000, B 0.000, C 0.000 }
gfCNCPoint1[25641] = {X 396.4173, Y 70.8229, Z -2.1667, A 0.000, B 0.000, C 0.000 }
gfCNCPoint1[25642] = {X 396.4160, Y 84.5909, Z -2.1667, A 0.000, B 0.000, C 0.000 }
gfCNCPoint1[25643] = {X 396.4157, Y 84.9469, Z -2.1667, A 0.000, B 0.000, C 0.000 }
gfCNCPoint1[25644] = {X 411.0610, Y 75.5672, Z -2.1667, A 0.000, B 0.000, C 0.000 }
gfCNCPoint1[25645] = {X 400.9149, Y 71.5862, Z -2.1667, A 0.000, B 0.000, C 0.000 }
gfCNCPoint1[25646] = {X 400.0767, Y 71.3060, Z -2.1667, A 0.000, B 0.000, C 0.000 }
gfCNCPoint1[25647] = {X 399.2139, Y 71.1146, Z -2.1667, A 0.000, B 0.000, C 0.000 }
gfCNCPoint1[25648] = {X 399.6108, Y 68.7477, Z -2.1667, A 0.000, B 0.000, C 0.000 }
gfCNCPoint1[25649] = {X 398.9927, Y 68.6622, Z -2.1667, A 0.000, B 0.000, C 0.000 }
gfCNCPoint1[25650] = {X 398.3706, Y 68.6123, Z -2.1667, A 0.000, B 0.000, C 0.000 }
gfCNCPoint1[25651] = {X 397.6036, Y 68.5669, Z -2.1667, A 0.000, B 0.000, C 0.000 }
gfCNCPoint1[25652] = {X 396.8425, Y 68.4609, Z -2.1667, A 0.000, B 0.000, C 0.000 }
gfCNCPoint1[25653] = {X 395.3921, Y 68.0818, Z -2.1667, A 0.000, B 0.000, C 0.000 }
gfCNCPoint1[25654] = {X 394.0176, Y 67.4833, Z -2.1667, A 0.000, B 0.000, C 0.000 }
gfCNCPoint1[25655] = {X 394.0160, Y 84.5982, Z -2.1667, A 0.000, B 0.000, C 0.000 }
gfCNCPoint1[25656] = {X 394.0164, Y 84.7638, Z -2.1667, A 0.000, B 0.000, C 0.000 }
gfCNCPoint1[25657] = {X 394.0158, Y 84.9295, Z -2.1667, A 0.000, B 0.000, C 0.000 }
gfCNCPoint1[25658] = {X 393.9652, Y 86.3343, Z -2.1667, A 0.000, B 0.000, C 0.000 }
gfCNCPoint1[25659] = {X 393.8337, Y 87.7339, Z -2.1667, A 0.000, B 0.000, C 0.000 }
gfCNCPoint1[25660] = {X 395.0693, Y 87.4787, Z -2.1667, A 0.000, B 0.000, C 0.000 }
gfCNCPoint1[25661] = {X 396.3275, Y 87.3863, Z -2.1667, A 0.000, B 0.000, C 0.000 }
gfCNCPoint1[25662] = {X 396.7226, Y 87.3730, Z -2.1667, A 0.000, B 0.000, C 0.000 }
gfCNCPoint1[25663] = {X 397.1171, Y 87.3477, Z -2.1667, A 0.000, B 0.000, C 0.000 }
gfCNCPoint1[25664] = {X 416.3166, Y 75.0513, Z -2.1667, A 0.000, B 0.000, C 0.000 }
gfCNCPoint1[25665] = {X 401.7936, Y 69.3529, Z -2.1667, A 0.000, B 0.000, C 0.000 }
gfCNCPoint1[25666] = {X 400.7180, Y 68.9933, Z -2.1667, A 0.000, B 0.000, C 0.000 }
gfCNCPoint1[25667] = {X 399.6108, Y 68.7477, Z -2.1667, A 0.000, B 0.000, C 0.000 }
gfCNCPoint1[25668] = {X 400.0077, Y 66.3807, Z -2.1667, A 0.000, B 0.000, C 0.000 }
gfCNCPoint1[25669] = {X 399.2317, Y 66.2740, Z -2.1667, A 0.000, B 0.000, C 0.000 }
gfCNCPoint1[25670] = {X 398.4508, Y 66.2133, Z -2.1667, A 0.000, B 0.000, C 0.000 }
gfCNCPoint1[25671] = {X 397.3061, Y 66.1057, Z -2.1667, A 0.000, B 0.000, C 0.000 }
gfCNCPoint1[25672] = {X 396.1927, Y 65.8192, Z -2.1667, A 0.000, B 0.000, C 0.000 }
gfCNCPoint1[25673] = {X 395.1382, Y 65.3610, Z -2.1667, A 0.000, B 0.000, C 0.000 }
gfCNCPoint1[25674] = {X 394.1691, Y 64.7425, Z -2.1667, A 0.000, B 0.000, C 0.000 }
gfCNCPoint1[25675] = {X 393.3094, Y 63.9792, Z -2.1667, A 0.000, B 0.000, C 0.000 }
gfCNCPoint1[25676] = {X 392.5118, Y 64.6966, Z -2.1667, A 0.000, B 0.000, C 0.000 }
gfCNCPoint1[25677] = {X 391.6178, Y 65.2894, Z -2.1667, A 0.000, B 0.000, C 0.000 }
gfCNCPoint1[25678] = {X 391.6159, Y 84.6059, Z -2.1667, A 0.000, B 0.000, C 0.000 }
gfCNCPoint1[25679] = {X 391.5796, Y 86.0260, Z -2.1667, A 0.000, B 0.000, C 0.000 }
gfCNCPoint1[25680] = {X 391.4517, Y 87.4408, Z -2.1667, A 0.000, B 0.000, C 0.000 }
gfCNCPoint1[25681] = {X 391.2275, Y 88.8723, Z -2.1667, A 0.000, B 0.000, C 0.000 }
gfCNCPoint1[25682] = {X 390.9096, Y 90.2858, Z -2.1667, A 0.000, B 0.000, C 0.000 }
gfCNCPoint1[25683] = {X 390.3336, Y 92.0498, Z -2.1667, A 0.000, B 0.000, C 0.000 }
gfCNCPoint1[25684] = {X 389.5422, Y 93.7282, Z -2.1667, A 0.000, B 0.000, C 0.000 }
gfCNCPoint1[25685] = {X 388.5478, Y 95.2949, Z -2.1667, A 0.000, B 0.000, C 0.000 }
gfCNCPoint1[25686] = {X 389.3447, Y 95.2949, Z -2.1667, A 0.000, B 0.000, C 0.000 }
gfCNCPoint1[25687] = {X 389.7639, Y 94.0858, Z -2.1667, A 0.000, B 0.000, C 0.000 }
gfCNCPoint1[25688] = {X 390.3884, Y 92.9687, Z -2.1667, A 0.000, B 0.000, C 0.000 }
gfCNCPoint1[25689] = {X 391.1988, Y 91.9783, Z -2.1667, A 0.000, B 0.000, C 0.000 }
gfCNCPoint1[25690] = {X 392.1701, Y 91.1451, Z -2.1667, A 0.000, B 0.000, C 0.000 }
gfCNCPoint1[25691] = {X 393.2724, Y 90.4948, Z -2.1667, A 0.000, B 0.000, C 0.000 }
gfCNCPoint1[25692] = {X 394.4715, Y 90.0477, Z -2.1667, A 0.000, B 0.000, C 0.000 }
gfCNCPoint1[25693] = {X 395.4059, Y 89.8549, Z -2.1667, A 0.000, B 0.000, C 0.000 }
gfCNCPoint1[25694] = {X 396.3575, Y 89.7861, Z -2.1667, A 0.000, B 0.000, C 0.000 }
gfCNCPoint1[25695] = {X 397.1497, Y 89.7493, Z -2.1667, A 0.000, B 0.000, C 0.000 }
gfCNCPoint1[25696] = {X 397.9389, Y 89.6714, Z -2.1667, A 0.000, B 0.000, C 0.000 }
gfCNCPoint1[25697] = {X 421.5723, Y 74.5353, Z -2.1667, A 0.000, B 0.000, C 0.000 }
gfCNCPoint1[25698] = {X 402.6722, Y 67.1195, Z -2.1667, A 0.000, B 0.000, C 0.000 }
gfCNCPoint1[25699] = {X 401.3593, Y 66.6805, Z -2.1667, A 0.000, B 0.000, C 0.000 }
gfCNCPoint1[25700] = {X 400.0077, Y 66.3807, Z -2.1667, A 0.000, B 0.000, C 0.000 }
gfCNCPoint1[25701] = {X 400.4046, Y 64.0138, Z -2.1667, A 0.000, B 0.000, C 0.000 }
gfCNCPoint1[25702] = {X 399.4656, Y 63.8853, Z -2.1667, A 0.000, B 0.000, C 0.000 }
gfCNCPoint1[25703] = {X 398.5205, Y 63.8139, Z -2.1667, A 0.000, B 0.000, C 0.000 }
gfCNCPoint1[25704] = {X 397.5547, Y 63.7099, Z -2.1667, A 0.000, B 0.000, C 0.000 }
gfCNCPoint1[25705] = {X 396.6287, Y 63.4166, Z -2.1667, A 0.000, B 0.000, C 0.000 }
gfCNCPoint1[25706] = {X 395.7791, Y 62.9458, Z -2.1667, A 0.000, B 0.000, C 0.000 }
gfCNCPoint1[25707] = {X 395.0396, Y 62.3159, Z -2.1667, A 0.000, B 0.000, C 0.000 }
gfCNCPoint1[25708] = {X 394.4659, Y 61.5933, Z -2.1667, A 0.000, B 0.000, C 0.000 }
gfCNCPoint1[25709] = {X 394.0385, Y 60.7756, Z -2.1667, A 0.000, B 0.000, C 0.000 }
gfCNCPoint1[25710] = {X 393.7727, Y 59.8921, Z -2.1667, A 0.000, B 0.000, C 0.000 }
gfCNCPoint1[25711] = {X 393.6779, Y 58.9744, Z -2.1667, A 0.000, B 0.000, C 0.000 }
gfCNCPoint1[25712] = {X 393.6777, Y 58.0000, Z -2.1667, A 0.000, B 0.000, C 0.000 }
gfCNCPoint1[25713] = {X 393.7668, Y 57.0718, Z -2.1667, A 0.000, B 0.000, C 0.000 }
gfCNCPoint1[25714] = {X 394.0309, Y 56.1774, Z -2.1667, A 0.000, B 0.000, C 0.000 }
gfCNCPoint1[25715] = {X 394.4602, Y 55.3496, Z -2.1667, A 0.000, B 0.000, C 0.000 }
gfCNCPoint1[25716] = {X 395.0391, Y 54.6186, Z -2.1667, A 0.000, B 0.000, C 0.000 }
gfCNCPoint1[25717] = {X 395.7864, Y 53.9833, Z -2.1667, A 0.000, B 0.000, C 0.000 }
gfCNCPoint1[25718] = {X 396.6455, Y 53.5102, Z -2.1667, A 0.000, B 0.000, C 0.000 }
gfCNCPoint1[25719] = {X 397.5819, Y 53.2186, Z -2.1667, A 0.000, B 0.000, C 0.000 }
gfCNCPoint1[25720] = {X 398.5577, Y 53.1200, Z -2.1667, A 0.000, B 0.000, C 0.000 }
gfCNCPoint1[25721] = {X 419.4886, Y 53.1200, Z -2.1667, A 0.000, B 0.000, C 0.000 }
gfCNCPoint1[25722] = {X 420.5535, Y 53.2376, Z -2.1667, A 0.000, B 0.000, C 0.000 }
gfCNCPoint1[25723] = {X 421.5670, Y 53.5847, Z -2.1667, A 0.000, B 0.000, C 0.000 }
gfCNCPoint1[25724] = {X 422.4804, Y 54.1447, Z -2.1667, A 0.000, B 0.000, C 0.000 }
gfCNCPoint1[25725] = {X 423.2496, Y 54.8904, Z -2.1667, A 0.000, B 0.000, C 0.000 }
gfCNCPoint1[25726] = {X 423.8375, Y 55.7860, Z -2.1667, A 0.000, B 0.000, C 0.000 }
gfCNCPoint1[25727] = {X 424.2158, Y 56.7883, Z -2.1667, A 0.000, B 0.000, C 0.000 }
gfCNCPoint1[25728] = {X 424.3663, Y 57.8490, Z -2.1667, A 0.000, B 0.000, C 0.000 }
gfCNCPoint1[25729] = {X 429.8190, Y 59.9742, Z -2.1667, A 0.000, B 0.000, C 0.000 }
gfCNCPoint1[25730] = {X 457.3009, Y 70.8775, Z -2.1667, A 0.000, B 0.000, C 0.000 }
gfCNCPoint1[25731] = {X 457.2999, Y 63.6743, Z -2.1667, A 0.000, B 0.000, C 0.000 }
gfCNCPoint1[25732] = {X 456.2915, Y 63.3060, Z -2.1667, A 0.000, B 0.000, C 0.000 }
gfCNCPoint1[25733] = {X 455.3880, Y 62.7261, Z -2.1667, A 0.000, B 0.000, C 0.000 }
gfCNCPoint1[25734] = {X 454.6332, Y 61.9628, Z -2.1667, A 0.000, B 0.000, C 0.000 }
gfCNCPoint1[25735] = {X 454.0636, Y 61.0528, Z -2.1667, A 0.000, B 0.000, C 0.000 }
gfCNCPoint1[25736] = {X 453.7067, Y 60.0404, Z -2.1667, A 0.000, B 0.000, C 0.000 }
gfCNCPoint1[25737] = {X 453.5798, Y 58.9744, Z -2.1667, A 0.000, B 0.000, C 0.000 }
gfCNCPoint1[25738] = {X 453.5796, Y 58.0000, Z -2.1667, A 0.000, B 0.000, C 0.000 }
gfCNCPoint1[25739] = {X 453.6734, Y 57.0480, Z -2.1667, A 0.000, B 0.000, C 0.000 }
gfCNCPoint1[25740] = {X 453.9511, Y 56.1325, Z -2.1667, A 0.000, B 0.000, C 0.000 }
gfCNCPoint1[25741] = {X 454.4020, Y 55.2888, Z -2.1667, A 0.000, B 0.000, C 0.000 }
gfCNCPoint1[25742] = {X 455.0089, Y 54.5493, Z -2.1667, A 0.000, B 0.000, C 0.000 }
gfCNCPoint1[25743] = {X 455.7484, Y 53.9424, Z -2.1667, A 0.000, B 0.000, C 0.000 }
gfCNCPoint1[25744] = {X 456.5921, Y 53.4915, Z -2.1667, A 0.000, B 0.000, C 0.000 }
gfCNCPoint1[25745] = {X 457.5076, Y 53.2138, Z -2.1667, A 0.000, B 0.000, C 0.000 }
gfCNCPoint1[25746] = {X 458.4596, Y 53.1200, Z -2.1667, A 0.000, B 0.000, C 0.000 }
gfCNCPoint1[25747] = {X 475.0000, Y 53.1200, Z -2.1667, A 0.000, B 0.000, C 0.000 }
gfCNCPoint1[25748] = {X 475.9520, Y 53.2138, Z -2.1667, A 0.000, B 0.000, C 0.000 }
gfCNCPoint1[25749] = {X 476.8675, Y 53.4915, Z -2.1667, A 0.000, B 0.000, C 0.000 }
gfCNCPoint1[25750] = {X 477.7112, Y 53.9424, Z -2.1667, A 0.000, B 0.000, C 0.000 }
gfCNCPoint1[25751] = {X 478.4507, Y 54.5493, Z -2.1667, A 0.000, B 0.000, C 0.000 }
gfCNCPoint1[25752] = {X 479.0576, Y 55.2888, Z -2.1667, A 0.000, B 0.000, C 0.000 }
gfCNCPoint1[25753] = {X 479.5085, Y 56.1325, Z -2.1667, A 0.000, B 0.000, C 0.000 }
gfCNCPoint1[25754] = {X 479.7862, Y 57.0480, Z -2.1667, A 0.000, B 0.000, C 0.000 }
gfCNCPoint1[25755] = {X 479.8800, Y 58.0000, Z -2.1667, A 0.000, B 0.000, C 0.000 }
gfCNCPoint1[25756] = {X 479.8798, Y 58.9744, Z -2.1667, A 0.000, B 0.000, C 0.000 }
gfCNCPoint1[25757] = {X 479.7529, Y 60.0404, Z -2.1667, A 0.000, B 0.000, C 0.000 }
gfCNCPoint1[25758] = {X 479.3960, Y 61.0529, Z -2.1667, A 0.000, B 0.000, C 0.000 }
gfCNCPoint1[25759] = {X 478.8263, Y 61.9629, Z -2.1667, A 0.000, B 0.000, C 0.000 }
gfCNCPoint1[25760] = {X 478.0714, Y 62.7262, Z -2.1667, A 0.000, B 0.000, C 0.000 }
gfCNCPoint1[25761] = {X 477.1679, Y 63.3061, Z -2.1667, A 0.000, B 0.000, C 0.000 }
gfCNCPoint1[25762] = {X 476.1595, Y 63.6743, Z -2.1667, A 0.000, B 0.000, C 0.000 }
gfCNCPoint1[25763] = {X 476.1599, Y 92.3323, Z -2.1667, A 0.000, B 0.000, C 0.000 }
gfCNCPoint1[25764] = {X 476.3625, Y 92.3916, Z -2.1667, A 0.000, B 0.000, C 0.000 }
gfCNCPoint1[25765] = {X 476.5636, Y 92.4560, Z -2.1667, A 0.000, B 0.000, C 0.000 }
gfCNCPoint1[25766] = {X 477.4816, Y 92.8730, Z -2.1667, A 0.000, B 0.000, C 0.000 }
gfCNCPoint1[25767] = {X 478.2936, Y 93.4706, Z -2.1667, A 0.000, B 0.000, C 0.000 }
gfCNCPoint1[25768] = {X 478.9646, Y 94.2230, Z -2.1667, A 0.000, B 0.000, C 0.000 }
gfCNCPoint1[25769] = {X 479.4657, Y 95.0978, Z -2.1667, A 0.000, B 0.000, C 0.000 }
gfCNCPoint1[25770] = {X 479.7753, Y 96.0573, Z -2.1667, A 0.000, B 0.000, C 0.000 }
gfCNCPoint1[25771] = {X 479.8800, Y 97.0600, Z -2.1667, A 0.000, B 0.000, C 0.000 }
gfCNCPoint1[25772] = {X 479.8800, Y 97.6949, Z -2.1667, A 0.000, B 0.000, C 0.000 }
gfCNCPoint1[25773] = {X 479.4000, Y 97.6949, Z -2.1667, A 0.000, B 0.000, C 0.000 }
gfCNCPoint1[25774] = {X 479.4000, Y 98.0000, Z -2.1667, A 0.000, B 0.000, C 0.000 }
gfCNCPoint1[25775] = {X 479.2897, Y 98.9791, Z -2.1667, A 0.000, B 0.000, C 0.000 }
gfCNCPoint1[25776] = {X 478.9643, Y 99.9091, Z -2.1667, A 0.000, B 0.000, C 0.000 }
gfCNCPoint1[25777] = {X 478.4401, Y 100.7434, Z -2.1667, A 0.000, B 0.000, C 0.000 }
gfCNCPoint1[25778] = {X 477.7434, Y 101.4401, Z -2.1667, A 0.000, B 0.000, C 0.000 }
gfCNCPoint1[25779] = {X 476.9091, Y 101.9643, Z -2.1667, A 0.000, B 0.000, C 0.000 }
gfCNCPoint1[25780] = {X 475.9791, Y 102.2897, Z -2.1667, A 0.000, B 0.000, C 0.000 }
gfCNCPoint1[25781] = {X 475.0000, Y 102.4000, Z -2.1667, A 0.000, B 0.000, C 0.000 }
gfCNCPoint1[25782] = {X 458.4596, Y 102.4000, Z -2.1667, A 0.000, B 0.000, C 0.000 }
gfCNCPoint1[25783] = {X 457.4805, Y 102.2897, Z -2.1667, A 0.000, B 0.000, C 0.000 }
gfCNCPoint1[25784] = {X 456.5505, Y 101.9643, Z -2.1667, A 0.000, B 0.000, C 0.000 }
gfCNCPoint1[25785] = {X 455.7162, Y 101.4401, Z -2.1667, A 0.000, B 0.000, C 0.000 }
gfCNCPoint1[25786] = {X 455.0195, Y 100.7434, Z -2.1667, A 0.000, B 0.000, C 0.000 }
gfCNCPoint1[25787] = {X 454.4953, Y 99.9091, Z -2.1667, A 0.000, B 0.000, C 0.000 }
gfCNCPoint1[25788] = {X 454.1699, Y 98.9791, Z -2.1667, A 0.000, B 0.000, C 0.000 }
gfCNCPoint1[25789] = {X 454.0596, Y 98.0000, Z -2.1667, A 0.000, B 0.000, C 0.000 }
gfCNCPoint1[25790] = {X 454.0596, Y 97.0659, Z -2.1667, A 0.000, B 0.000, C 0.000 }
gfCNCPoint1[25791] = {X 454.1492, Y 96.1826, Z -2.1667, A 0.000, B 0.000, C 0.000 }
gfCNCPoint1[25792] = {X 454.4143, Y 95.3353, Z -2.1667, A 0.000, B 0.000, C 0.000 }
gfCNCPoint1[25793] = {X 454.8440, Y 94.5584, Z -2.1667, A 0.000, B 0.000, C 0.000 }
gfCNCPoint1[25794] = {X 455.4210, Y 93.8836, Z -2.1667, A 0.000, B 0.000, C 0.000 }
gfCNCPoint1[25795] = {X 456.1217, Y 93.3384, Z -2.1667, A 0.000, B 0.000, C 0.000 }
gfCNCPoint1[25796] = {X 456.9176, Y 92.9450, Z -2.1667, A 0.000, B 0.000, C 0.000 }
gfCNCPoint1[25797] = {X 457.7763, Y 92.7193, Z -2.1667, A 0.000, B 0.000, C 0.000 }
gfCNCPoint1[25798] = {X 457.7763, Y 85.6495, Z -2.1667, A 0.000, B 0.000, C 0.000 }
gfCNCPoint1[25799] = {X 444.8672, Y 80.5891, Z -2.1667, A 0.000, B 0.000, C 0.000 }
gfCNCPoint1[25800] = {X 420.1031, Y 96.6313, Z -2.1667, A 0.000, B 0.000, C 0.000 }
gfCNCPoint1[25801] = {X 420.1067, Y 97.0659, Z -2.1667, A 0.000, B 0.000, C 0.000 }
gfCNCPoint1[25802] = {X 420.1067, Y 98.0000, Z -2.1667, A 0.000, B 0.000, C 0.000 }
gfCNCPoint1[25803] = {X 419.9964, Y 98.9791, Z -2.1667, A 0.000, B 0.000, C 0.000 }
gfCNCPoint1[25804] = {X 419.6710, Y 99.9091, Z -2.1667, A 0.000, B 0.000, C 0.000 }
gfCNCPoint1[25805] = {X 419.1468, Y 100.7434, Z -2.1667, A 0.000, B 0.000, C 0.000 }
gfCNCPoint1[25806] = {X 418.4501, Y 101.4401, Z -2.1667, A 0.000, B 0.000, C 0.000 }
gfCNCPoint1[25807] = {X 417.6158, Y 101.9643, Z -2.1667, A 0.000, B 0.000, C 0.000 }
gfCNCPoint1[25808] = {X 416.6858, Y 102.2897, Z -2.1667, A 0.000, B 0.000, C 0.000 }
gfCNCPoint1[25809] = {X 415.7067, Y 102.4000, Z -2.1667, A 0.000, B 0.000, C 0.000 }
gfCNCPoint1[25810] = {X 396.4059, Y 102.4000, Z -2.1667, A 0.000, B 0.000, C 0.000 }
gfCNCPoint1[25811] = {X 395.4269, Y 102.2897, Z -2.1667, A 0.000, B 0.000, C 0.000 }
gfCNCPoint1[25812] = {X 394.4969, Y 101.9643, Z -2.1667, A 0.000, B 0.000, C 0.000 }
gfCNCPoint1[25813] = {X 393.6626, Y 101.4401, Z -2.1667, A 0.000, B 0.000, C 0.000 }
gfCNCPoint1[25814] = {X 392.9659, Y 100.7434, Z -2.1667, A 0.000, B 0.000, C 0.000 }
gfCNCPoint1[25815] = {X 392.4417, Y 99.9091, Z -2.1667, A 0.000, B 0.000, C 0.000 }
gfCNCPoint1[25816] = {X 392.1163, Y 98.9791, Z -2.1667, A 0.000, B 0.000, C 0.000 }
gfCNCPoint1[25817] = {X 392.0059, Y 98.0000, Z -2.1667, A 0.000, B 0.000, C 0.000 }
gfCNCPoint1[25818] = {X 392.0059, Y 97.0659, Z -2.1667, A 0.000, B 0.000, C 0.000 }
gfCNCPoint1[25819] = {X 392.1157, Y 96.0891, Z -2.1667, A 0.000, B 0.000, C 0.000 }
gfCNCPoint1[25820] = {X 392.4396, Y 95.1611, Z -2.1667, A 0.000, B 0.000, C 0.000 }
gfCNCPoint1[25821] = {X 392.9615, Y 94.3281, Z -2.1667, A 0.000, B 0.000, C 0.000 }
gfCNCPoint1[25822] = {X 393.6552, Y 93.6318, Z -2.1667, A 0.000, B 0.000, C 0.000 }
gfCNCPoint1[25823] = {X 394.4862, Y 93.1068, Z -2.1667, A 0.000, B 0.000, C 0.000 }
gfCNCPoint1[25824] = {X 395.4130, Y 92.7794, Z -2.1667, A 0.000, B 0.000, C 0.000 }
gfCNCPoint1[25825] = {X 396.3894, Y 92.6660, Z -2.1667, A 0.000, B 0.000, C 0.000 }
gfCNCPoint1[25826] = {X 397.3382, Y 92.6257, Z -2.1667, A 0.000, B 0.000, C 0.000 }
gfCNCPoint1[25827] = {X 398.2836, Y 92.5359, Z -2.1667, A 0.000, B 0.000, C 0.000 }
gfCNCPoint1[25828] = {X 398.9174, Y 92.3823, Z -2.1667, A 0.000, B 0.000, C 0.000 }
gfCNCPoint1[25829] = {X 399.5010, Y 92.0909, Z -2.1667, A 0.000, B 0.000, C 0.000 }
gfCNCPoint1[25830] = {X 405.1777, Y 88.4328, Z -2.1667, A 0.000, B 0.000, C 0.000 }
gfCNCPoint1[25831] = {X 427.8798, Y 73.9164, Z -2.1667, A 0.000, B 0.000, C 0.000 }
gfCNCPoint1[25832] = {X 403.7262, Y 64.4393, Z -2.1667, A 0.000, B 0.000, C 0.000 }
gfCNCPoint1[25833] = {X 402.0392, Y 63.8807, Z -2.1667, A 0.000, B 0.000, C 0.000 }
gfCNCPoint1[25834] = {X 400.3011, Y 63.5108, Z -2.1667, A 0.000, B 0.000, C 0.000 }
gfCNCPoint1[25835] = {X 398.5329, Y 63.3340, Z -2.1667, A 0.000, B 0.000, C 0.000 }
gfCNCPoint1[25836] = {X 397.5579, Y 63.2190, Z -2.1667, A 0.000, B 0.000, C 0.000 }
gfCNCPoint1[25837] = {X 396.6327, Y 62.8906, Z -2.1667, A 0.000, B 0.000, C 0.000 }
gfCNCPoint1[25838] = {X 395.8033, Y 62.3653, Z -2.1667, A 0.000, B 0.000, C 0.000 }
gfCNCPoint1[25839] = {X 395.1110, Y 61.6691, Z -2.1667, A 0.000, B 0.000, C 0.000 }
gfCNCPoint1[25840] = {X 394.5904, Y 60.8367, Z -2.1667, A 0.000, B 0.000, C 0.000 }
gfCNCPoint1[25841] = {X 394.2672, Y 59.9097, Z -2.1667, A 0.000, B 0.000, C 0.000 }
gfCNCPoint1[25842] = {X 394.1577, Y 58.9340, Z -2.1667, A 0.000, B 0.000, C 0.000 }
gfCNCPoint1[25843] = {X 394.1577, Y 58.0000, Z -2.1667, A 0.000, B 0.000, C 0.000 }
gfCNCPoint1[25844] = {X 394.2680, Y 57.0209, Z -2.1667, A 0.000, B 0.000, C 0.000 }
gfCNCPoint1[25845] = {X 394.5935, Y 56.0909, Z -2.1667, A 0.000, B 0.000, C 0.000 }
gfCNCPoint1[25846] = {X 395.1177, Y 55.2566, Z -2.1667, A 0.000, B 0.000, C 0.000 }
gfCNCPoint1[25847] = {X 395.8144, Y 54.5599, Z -2.1667, A 0.000, B 0.000, C 0.000 }
gfCNCPoint1[25848] = {X 396.6486, Y 54.0357, Z -2.1667, A 0.000, B 0.000, C 0.000 }
gfCNCPoint1[25849] = {X 397.5786, Y 53.7103, Z -2.1667, A 0.000, B 0.000, C 0.000 }
gfCNCPoint1[25850] = {X 398.5577, Y 53.6000, Z -2.1667, A 0.000, B 0.000, C 0.000 }
gfCNCPoint1[25851] = {X 419.4886, Y 53.6000, Z -2.1667, A 0.000, B 0.000, C 0.000 }
gfCNCPoint1[25852] = {X 420.4677, Y 53.7103, Z -2.1667, A 0.000, B 0.000, C 0.000 }
gfCNCPoint1[25853] = {X 421.3977, Y 54.0357, Z -2.1667, A 0.000, B 0.000, C 0.000 }
gfCNCPoint1[25854] = {X 422.2320, Y 54.5599, Z -2.1667, A 0.000, B 0.000, C 0.000 }
gfCNCPoint1[25855] = {X 422.9287, Y 55.2566, Z -2.1667, A 0.000, B 0.000, C 0.000 }
gfCNCPoint1[25856] = {X 423.4529, Y 56.0909, Z -2.1667, A 0.000, B 0.000, C 0.000 }
gfCNCPoint1[25857] = {X 423.7783, Y 57.0209, Z -2.1667, A 0.000, B 0.000, C 0.000 }
gfCNCPoint1[25858] = {X 423.8886, Y 58.0000, Z -2.1667, A 0.000, B 0.000, C 0.000 }
gfCNCPoint1[25859] = {X 423.8886, Y 58.1780, Z -2.1667, A 0.000, B 0.000, C 0.000 }
gfCNCPoint1[25860] = {X 429.6420, Y 60.4204, Z -2.1667, A 0.000, B 0.000, C 0.000 }
gfCNCPoint1[25861] = {X 457.7810, Y 71.5844, Z -2.1667, A 0.000, B 0.000, C 0.000 }
gfCNCPoint1[25862] = {X 457.7798, Y 63.2812, Z -2.1667, A 0.000, B 0.000, C 0.000 }
gfCNCPoint1[25863] = {X 456.9205, Y 63.0561, Z -2.1667, A 0.000, B 0.000, C 0.000 }
gfCNCPoint1[25864] = {X 456.1239, Y 62.6629, Z -2.1667, A 0.000, B 0.000, C 0.000 }
gfCNCPoint1[25865] = {X 455.4225, Y 62.1178, Z -2.1667, A 0.000, B 0.000, C 0.000 }
gfCNCPoint1[25866] = {X 454.8449, Y 61.4428, Z -2.1667, A 0.000, B 0.000, C 0.000 }
gfCNCPoint1[25867] = {X 454.4146, Y 60.6656, Z -2.1667, A 0.000, B 0.000, C 0.000 }
gfCNCPoint1[25868] = {X 454.1493, Y 59.8179, Z -2.1667, A 0.000, B 0.000, C 0.000 }
gfCNCPoint1[25869] = {X 454.0596, Y 58.9340, Z -2.1667, A 0.000, B 0.000, C 0.000 }
gfCNCPoint1[25870] = {X 454.0596, Y 58.0000, Z -2.1667, A 0.000, B 0.000, C 0.000 }
gfCNCPoint1[25871] = {X 454.1699, Y 57.0209, Z -2.1667, A 0.000, B 0.000, C 0.000 }
gfCNCPoint1[25872] = {X 454.4953, Y 56.0909, Z -2.1667, A 0.000, B 0.000, C 0.000 }
gfCNCPoint1[25873] = {X 455.0195, Y 55.2566, Z -2.1667, A 0.000, B 0.000, C 0.000 }
gfCNCPoint1[25874] = {X 455.7162, Y 54.5599, Z -2.1667, A 0.000, B 0.000, C 0.000 }
gfCNCPoint1[25875] = {X 456.5505, Y 54.0357, Z -2.1667, A 0.000, B 0.000, C 0.000 }
gfCNCPoint1[25876] = {X 457.4805, Y 53.7103, Z -2.1667, A 0.000, B 0.000, C 0.000 }
gfCNCPoint1[25877] = {X 458.4596, Y 53.6000, Z -2.1667, A 0.000, B 0.000, C 0.000 }
gfCNCPoint1[25878] = {X 475.0000, Y 53.6000, Z -2.1667, A 0.000, B 0.000, C 0.000 }
gfCNCPoint1[25879] = {X 475.9791, Y 53.7103, Z -2.1667, A 0.000, B 0.000, C 0.000 }
gfCNCPoint1[25880] = {X 476.9091, Y 54.0357, Z -2.1667, A 0.000, B 0.000, C 0.000 }
gfCNCPoint1[25881] = {X 477.7434, Y 54.5599, Z -2.1667, A 0.000, B 0.000, C 0.000 }
gfCNCPoint1[25882] = {X 478.4401, Y 55.2566, Z -2.1667, A 0.000, B 0.000, C 0.000 }
gfCNCPoint1[25883] = {X 478.9643, Y 56.0909, Z -2.1667, A 0.000, B 0.000, C 0.000 }
gfCNCPoint1[25884] = {X 479.2897, Y 57.0209, Z -2.1667, A 0.000, B 0.000, C 0.000 }
gfCNCPoint1[25885] = {X 479.4000, Y 58.0000, Z -2.1667, A 0.000, B 0.000, C 0.000 }
gfCNCPoint1[25886] = {X 479.3998, Y 58.9704, Z -2.1667, A 0.000, B 0.000, C 0.000 }
gfCNCPoint1[25887] = {X 479.3040, Y 59.8484, Z -2.1667, A 0.000, B 0.000, C 0.000 }
gfCNCPoint1[25888] = {X 479.0346, Y 60.6896, Z -2.1667, A 0.000, B 0.000, C 0.000 }
gfCNCPoint1[25889] = {X 478.6027, Y 61.4600, Z -2.1667, A 0.000, B 0.000, C 0.000 }
gfCNCPoint1[25890] = {X 478.0257, Y 62.1286, Z -2.1667, A 0.000, B 0.000, C 0.000 }
gfCNCPoint1[25891] = {X 477.3267, Y 62.6686, Z -2.1667, A 0.000, B 0.000, C 0.000 }
gfCNCPoint1[25892] = {X 476.5340, Y 63.0580, Z -2.1667, A 0.000, B 0.000, C 0.000 }
gfCNCPoint1[25893] = {X 475.6795, Y 63.2813, Z -2.1667, A 0.000, B 0.000, C 0.000 }
gfCNCPoint1[25894] = {X 475.6799, Y 92.7050, Z -2.1667, A 0.000, B 0.000, C 0.000 }
gfCNCPoint1[25895] = {X 476.0482, Y 92.7995, Z -2.1667, A 0.000, B 0.000, C 0.000 }
gfCNCPoint1[25896] = {X 476.4116, Y 92.9113, Z -2.1667, A 0.000, B 0.000, C 0.000 }
gfCNCPoint1[25897] = {X 477.2387, Y 93.2870, Z -2.1667, A 0.000, B 0.000, C 0.000 }
gfCNCPoint1[25898] = {X 477.9704, Y 93.8255, Z -2.1667, A 0.000, B 0.000, C 0.000 }
gfCNCPoint1[25899] = {X 478.5751, Y 94.5035, Z -2.1667, A 0.000, B 0.000, C 0.000 }
gfCNCPoint1[25900] = {X 479.0267, Y 95.2919, Z -2.1667, A 0.000, B 0.000, C 0.000 }
gfCNCPoint1[25901] = {X 479.3057, Y 96.1565, Z -2.1667, A 0.000, B 0.000, C 0.000 }
gfCNCPoint1[25902] = {X 479.4000, Y 97.0600, Z -2.1667, A 0.000, B 0.000, C 0.000 }
gfCNCPoint1[25903] = {X 479.4000, Y 97.6949, Z -2.1667, A 0.000, B 0.000, C 0.000 }
gfCNCPoint1[25904] = {X 479.8800, Y 97.6949, Z -2.1667, A 0.000, B 0.000, C 0.000 }
gfCNCPoint1[25905] = {X 507.6819, Y 97.6949, Z -2.1667, A 0.000, B 0.000, C 0.000 }
gfCNCPoint1[25906] = {X 507.6819, Y 100.0949, Z -2.1667, A 0.000, B 0.000, C 0.000 }
gfCNCPoint1[25907] = {X 600.0148, Y 100.0949, Z -2.1667, A 0.000, B 0.000, C 0.000 }
gfCNCPoint1[25908] = {X 600.0671, Y 100.0697, Z -2.1667, A 0.000, B 0.000, C 0.000 }
gfCNCPoint1[25909] = {X 600.0948, Y 100.0187, Z -2.1667, A 0.000, B 0.000, C 0.000 }
gfCNCPoint1[25910] = {X 600.0965, Y 99.1431, Z -2.1667, A 0.000, B 0.000, C 0.000 }
gfCNCPoint1[25911] = {X 600.0965, Y 49.8790, Z -2.1667, A 0.000, B 0.000, C 0.000 }
gfCNCPoint1[25912] = {X 601.1111, Y 49.7518, Z -2.1667, A 0.000, B 0.000, C 0.000 }
gfCNCPoint1[25913] = {X 602.0768, Y 49.4160, Z -2.1667, A 0.000, B 0.000, C 0.000 }
gfCNCPoint1[25914] = {X 602.9515, Y 48.8863, Z -2.1667, A 0.000, B 0.000, C 0.000 }
gfCNCPoint1[25915] = {X 603.6965, Y 48.1860, Z -2.1667, A 0.000, B 0.000, C 0.000 }
gfCNCPoint1[25916] = {X 603.6965, Y 47.3866, Z -2.1667, A 0.000, B 0.000, C 0.000 }
gfCNCPoint1[25917] = {X 603.1502, Y 48.0718, Z -2.1667, A 0.000, B 0.000, C 0.000 }
gfCNCPoint1[25918] = {X 602.4789, Y 48.6352, Z -2.1667, A 0.000, B 0.000, C 0.000 }
gfCNCPoint1[25919] = {X 601.7094, Y 49.0544, Z -2.1667, A 0.000, B 0.000, C 0.000 }
gfCNCPoint1[25920] = {X 600.8720, Y 49.3127, Z -2.1667, A 0.000, B 0.000, C 0.000 }
gfCNCPoint1[25921] = {X 600.0000, Y 49.4000, Z -2.1667, A 0.000, B 0.000, C 0.000 }
gfCNCPoint1[25922] = {X 593.5565, Y 49.4000, Z -2.1667, A 0.000, B 0.000, C 0.000 }
gfCNCPoint1[25923] = {X 592.5988, Y 49.2945, Z -2.1667, A 0.000, B 0.000, C 0.000 }
gfCNCPoint1[25924] = {X 591.6870, Y 48.9831, Z -2.1667, A 0.000, B 0.000, C 0.000 }
gfCNCPoint1[25925] = {X 590.8648, Y 48.4806, Z -2.1667, A 0.000, B 0.000, C 0.000 }
gfCNCPoint1[25926] = {X 590.1717, Y 47.8112, Z -2.1667, A 0.000, B 0.000, C 0.000 }
gfCNCPoint1[25927] = {X 589.6410, Y 47.0071, Z -2.1667, A 0.000, B 0.000, C 0.000 }
gfCNCPoint1[25928] = {X 589.3741, Y 46.3664, Z -2.1667, A 0.000, B 0.000, C 0.000 }
gfCNCPoint1[25929] = {X 589.2113, Y 45.6918, Z -2.1667, A 0.000, B 0.000, C 0.000 }
gfCNCPoint1[25930] = {X 589.1565, Y 45.0000, Z -2.1667, A 0.000, B 0.000, C 0.000 }
gfCNCPoint1[25931] = {X 589.1565, Y 44.0639, Z -2.1667, A 0.000, B 0.000, C 0.000 }
gfCNCPoint1[25932] = {X 589.2613, Y 43.1277, Z -2.1667, A 0.000, B 0.000, C 0.000 }
gfCNCPoint1[25933] = {X 589.5611, Y 42.2346, Z -2.1667, A 0.000, B 0.000, C 0.000 }
gfCNCPoint1[25934] = {X 590.0424, Y 41.4248, Z -2.1667, A 0.000, B 0.000, C 0.000 }
gfCNCPoint1[25935] = {X 590.6836, Y 40.7346, Z -2.1667, A 0.000, B 0.000, C 0.000 }
gfCNCPoint1[25936] = {X 590.6851, Y 40.3069, Z -2.1667, A 0.000, B 0.000, C 0.000 }
gfCNCPoint1[25937] = {X 590.6841, Y 35.2162, Z -2.1667, A 0.000, B 0.000, C 0.000 }
gfCNCPoint1[25938] = {X 590.6838, Y 33.9388, Z -2.1667, A 0.000, B 0.000, C 0.000 }
gfCNCPoint1[25939] = {X 585.5192, Y 46.6830, Z -2.1667, A 0.000, B 0.000, C 0.000 }
gfCNCPoint1[25940] = {X 585.4476, Y 46.8466, Z -2.1667, A 0.000, B 0.000, C 0.000 }
gfCNCPoint1[25941] = {X 585.3694, Y 47.0071, Z -2.1667, A 0.000, B 0.000, C 0.000 }
gfCNCPoint1[25942] = {X 584.8417, Y 47.8075, Z -2.1667, A 0.000, B 0.000, C 0.000 }
gfCNCPoint1[25943] = {X 584.1532, Y 48.4747, Z -2.1667, A 0.000, B 0.000, C 0.000 }
gfCNCPoint1[25944] = {X 583.3365, Y 48.9769, Z -2.1667, A 0.000, B 0.000, C 0.000 }
gfCNCPoint1[25945] = {X 582.4111, Y 49.2946, Z -2.1667, A 0.000, B 0.000, C 0.000 }
gfCNCPoint1[25946] = {X 581.4384, Y 49.4000, Z -2.1667, A 0.000, B 0.000, C 0.000 }
gfCNCPoint1[25947] = {X 580.4664, Y 49.2878, Z -2.1667, A 0.000, B 0.000, C 0.000 }
gfCNCPoint1[25948] = {X 579.5433, Y 48.9635, Z -2.1667, A 0.000, B 0.000, C 0.000 }
gfCNCPoint1[25949] = {X 578.7146, Y 48.4433, Z -2.1667, A 0.000, B 0.000, C 0.000 }
gfCNCPoint1[25950] = {X 578.0214, Y 47.7529, Z -2.1667, A 0.000, B 0.000, C 0.000 }
gfCNCPoint1[25951] = {X 577.4979, Y 46.9263, Z -2.1667, A 0.000, B 0.000, C 0.000 }
gfCNCPoint1[25952] = {X 577.4375, Y 46.7968, Z -2.1667, A 0.000, B 0.000, C 0.000 }
gfCNCPoint1[25953] = {X 577.3813, Y 46.6655, Z -2.1667, A 0.000, B 0.000, C 0.000 }
gfCNCPoint1[25954] = {X 572.5780, Y 34.9201, Z -2.1667, A 0.000, B 0.000, C 0.000 }
gfCNCPoint1[25955] = {X 572.0979, Y 33.7462, Z -2.1667, A 0.000, B 0.000, C 0.000 }
gfCNCPoint1[25956] = {X 572.0983, Y 40.7324, Z -2.1667, A 0.000, B 0.000, C 0.000 }
gfCNCPoint1[25957] = {X 572.7432, Y 41.4216, Z -2.1667, A 0.000, B 0.000, C 0.000 }
gfCNCPoint1[25958] = {X 573.2262, Y 42.2324, Z -2.1667, A 0.000, B 0.000, C 0.000 }
gfCNCPoint1[25959] = {X 573.5252, Y 43.1276, Z -2.1667, A 0.000, B 0.000, C 0.000 }
gfCNCPoint1[25960] = {X 573.6264, Y 44.0660, Z -2.1667, A 0.000, B 0.000, C 0.000 }
gfCNCPoint1[25961] = {X 573.6264, Y 45.0000, Z -2.1667, A 0.000, B 0.000, C 0.000 }
gfCNCPoint1[25962] = {X 573.5140, Y 45.9884, Z -2.1667, A 0.000, B 0.000, C 0.000 }
gfCNCPoint1[25963] = {X 573.1824, Y 46.9263, Z -2.1667, A 0.000, B 0.000, C 0.000 }
gfCNCPoint1[25964] = {X 572.6569, Y 47.7553, Z -2.1667, A 0.000, B 0.000, C 0.000 }
gfCNCPoint1[25965] = {X 571.9608, Y 48.4472, Z -2.1667, A 0.000, B 0.000, C 0.000 }
gfCNCPoint1[25966] = {X 571.1286, Y 48.9676, Z -2.1667, A 0.000, B 0.000, C 0.000 }
gfCNCPoint1[25967] = {X 570.2018, Y 49.2905, Z -2.1667, A 0.000, B 0.000, C 0.000 }
gfCNCPoint1[25968] = {X 569.2264, Y 49.4000, Z -2.1667, A 0.000, B 0.000, C 0.000 }
gfCNCPoint1[25969] = {X 562.4443, Y 49.4000, Z -2.1667, A 0.000, B 0.000, C 0.000 }
gfCNCPoint1[25970] = {X 561.4652, Y 49.2897, Z -2.1667, A 0.000, B 0.000, C 0.000 }
gfCNCPoint1[25971] = {X 560.5352, Y 48.9643, Z -2.1667, A 0.000, B 0.000, C 0.000 }
gfCNCPoint1[25972] = {X 559.7009, Y 48.4401, Z -2.1667, A 0.000, B 0.000, C 0.000 }
gfCNCPoint1[25973] = {X 559.0042, Y 47.7434, Z -2.1667, A 0.000, B 0.000, C 0.000 }
gfCNCPoint1[25974] = {X 558.4800, Y 46.9091, Z -2.1667, A 0.000, B 0.000, C 0.000 }
gfCNCPoint1[25975] = {X 558.1546, Y 45.9791, Z -2.1667, A 0.000, B 0.000, C 0.000 }
gfCNCPoint1[25976] = {X 558.0443, Y 45.0000, Z -2.1667, A 0.000, B 0.000, C 0.000 }
gfCNCPoint1[25977] = {X 558.0443, Y 44.0641, Z -2.1667, A 0.000, B 0.000, C 0.000 }
gfCNCPoint1[25978] = {X 558.1489, Y 43.1276, Z -2.1667, A 0.000, B 0.000, C 0.000 }
gfCNCPoint1[25979] = {X 558.4489, Y 42.2343, Z -2.1667, A 0.000, B 0.000, C 0.000 }
gfCNCPoint1[25980] = {X 558.9307, Y 41.4245, Z -2.1667, A 0.000, B 0.000, C 0.000 }
gfCNCPoint1[25981] = {X 559.5727, Y 40.7346, Z -2.1667, A 0.000, B 0.000, C 0.000 }
gfCNCPoint1[25982] = {X 559.5727, Y 9.2678, Z -2.1667, A 0.000, B 0.000, C 0.000 }
gfCNCPoint1[25983] = {X 558.9277, Y 8.5786, Z -2.1667, A 0.000, B 0.000, C 0.000 }
gfCNCPoint1[25984] = {X 558.4446, Y 7.7677, Z -2.1667, A 0.000, B 0.000, C 0.000 }
gfCNCPoint1[25985] = {X 558.1455, Y 6.8724, Z -2.1667, A 0.000, B 0.000, C 0.000 }
gfCNCPoint1[25986] = {X 558.0443, Y 5.9339, Z -2.1667, A 0.000, B 0.000, C 0.000 }
gfCNCPoint1[25987] = {X 558.0443, Y 5.0000, Z -2.1667, A 0.000, B 0.000, C 0.000 }
gfCNCPoint1[25988] = {X 558.1353, Y 4.1097, Z -2.1667, A 0.000, B 0.000, C 0.000 }
gfCNCPoint1[25989] = {X 558.4046, Y 3.2562, Z -2.1667, A 0.000, B 0.000, C 0.000 }
gfCNCPoint1[25990] = {X 558.9155, Y 2.3718, Z -2.1667, A 0.000, B 0.000, C 0.000 }
gfCNCPoint1[25991] = {X 559.6165, Y 1.6290, Z -2.1667, A 0.000, B 0.000, C 0.000 }
gfCNCPoint1[25992] = {X 560.4700, Y 1.0678, Z -2.1667, A 0.000, B 0.000, C 0.000 }
gfCNCPoint1[25993] = {X 561.4298, Y 0.7186, Z -2.1667, A 0.000, B 0.000, C 0.000 }
gfCNCPoint1[25994] = {X 562.4443, Y 0.6000, Z -2.1667, A 0.000, B 0.000, C 0.000 }
gfCNCPoint1[25995] = {X 570.9376, Y 0.6000, Z -2.1667, A 0.000, B 0.000, C 0.000 }
gfCNCPoint1[25996] = {X 571.9520, Y 0.7186, Z -2.1667, A 0.000, B 0.000, C 0.000 }
gfCNCPoint1[25997] = {X 572.9119, Y 1.0678, Z -2.1667, A 0.000, B 0.000, C 0.000 }
gfCNCPoint1[25998] = {X 573.7653, Y 1.6290, Z -2.1667, A 0.000, B 0.000, C 0.000 }
gfCNCPoint1[25999] = {X 574.4664, Y 2.3718, Z -2.1667, A 0.000, B 0.000, C 0.000 }
gfCNCPoint1[26000] = {X 574.9773, Y 3.2562, Z -2.1667, A 0.000, B 0.000, C 0.000 }
gfCNCPoint1[26001] = {X 575.2317, Y 4.0407, Z -2.1667, A 0.000, B 0.000, C 0.000 }
gfCNCPoint1[26002] = {X 575.3353, Y 4.8590, Z -2.1667, A 0.000, B 0.000, C 0.000 }
gfCNCPoint1[26003] = {X 580.1328, Y 4.7051, Z -2.1667, A 0.000, B 0.000, C 0.000 }
gfCNCPoint1[26004] = {X 580.1364, Y 4.8525, Z -2.1667, A 0.000, B 0.000, C 0.000 }
gfCNCPoint1[26005] = {X 580.1376, Y 5.0000, Z -2.1667, A 0.000, B 0.000, C 0.000 }
gfCNCPoint1[26006] = {X 580.1376, Y 5.9338, Z -2.1667, A 0.000, B 0.000, C 0.000 }
gfCNCPoint1[26007] = {X 580.0683, Y 7.0606, Z -2.1667, A 0.000, B 0.000, C 0.000 }
gfCNCPoint1[26008] = {X 579.8616, Y 8.1703, Z -2.1667, A 0.000, B 0.000, C 0.000 }
gfCNCPoint1[26009] = {X 581.1998, Y 11.4550, Z -2.1667, A 0.000, B 0.000, C 0.000 }
gfCNCPoint1[26010] = {X 582.6185, Y 7.9852, Z -2.1667, A 0.000, B 0.000, C 0.000 }
gfCNCPoint1[26011] = {X 582.4489, Y 6.9999, Z -2.1667, A 0.000, B 0.000, C 0.000 }
gfCNCPoint1[26012] = {X 582.3872, Y 6.0020, Z -2.1667, A 0.000, B 0.000, C 0.000 }
gfCNCPoint1[26013] = {X 582.3870, Y 5.0000, Z -2.1667, A 0.000, B 0.000, C 0.000 }
gfCNCPoint1[26014] = {X 582.3881, Y 4.8525, Z -2.1667, A 0.000, B 0.000, C 0.000 }
gfCNCPoint1[26015] = {X 582.3917, Y 4.7051, Z -2.1667, A 0.000, B 0.000, C 0.000 }
gfCNCPoint1[26016] = {X 580.1328, Y 4.7051, Z -2.1667, A 0.000, B 0.000, C 0.000 }
gfCNCPoint1[26017] = {X 577.7341, Y 4.7820, Z -2.1667, A 0.000, B 0.000, C 0.000 }
gfCNCPoint1[26018] = {X 577.7367, Y 4.8910, Z -2.1667, A 0.000, B 0.000, C 0.000 }
gfCNCPoint1[26019] = {X 577.7376, Y 5.0000, Z -2.1667, A 0.000, B 0.000, C 0.000 }
gfCNCPoint1[26020] = {X 577.7376, Y 5.9339, Z -2.1667, A 0.000, B 0.000, C 0.000 }
gfCNCPoint1[26021] = {X 577.6317, Y 7.1290, Z -2.1667, A 0.000, B 0.000, C 0.000 }
gfCNCPoint1[26022] = {X 577.3176, Y 8.2868, Z -2.1667, A 0.000, B 0.000, C 0.000 }
gfCNCPoint1[26023] = {X 581.1958, Y 17.8062, Z -2.1667, A 0.000, B 0.000, C 0.000 }
gfCNCPoint1[26024] = {X 585.1517, Y 8.1312, Z -2.1667, A 0.000, B 0.000, C 0.000 }
gfCNCPoint1[26025] = {X 584.8835, Y 7.0760, Z -2.1667, A 0.000, B 0.000, C 0.000 }
gfCNCPoint1[26026] = {X 584.7872, Y 5.9916, Z -2.1667, A 0.000, B 0.000, C 0.000 }
gfCNCPoint1[26027] = {X 584.7870, Y 5.0000, Z -2.1667, A 0.000, B 0.000, C 0.000 }
gfCNCPoint1[26028] = {X 584.7878, Y 4.8910, Z -2.1667, A 0.000, B 0.000, C 0.000 }
gfCNCPoint1[26029] = {X 584.7904, Y 4.7820, Z -2.1667, A 0.000, B 0.000, C 0.000 }
gfCNCPoint1[26030] = {X 584.9505, Y 3.5175, Z -2.1667, A 0.000, B 0.000, C 0.000 }
gfCNCPoint1[26031] = {X 585.3438, Y 2.3051, Z -2.1667, A 0.000, B 0.000, C 0.000 }
gfCNCPoint1[26032] = {X 577.1807, Y 2.3051, Z -2.1667, A 0.000, B 0.000, C 0.000 }
gfCNCPoint1[26033] = {X 577.5740, Y 3.5175, Z -2.1667, A 0.000, B 0.000, C 0.000 }
gfCNCPoint1[26034] = {X 577.7341, Y 4.7820, Z -2.1667, A 0.000, B 0.000, C 0.000 }
gfCNCPoint1[26035] = {X 575.3353, Y 4.8590, Z -2.1667, A 0.000, B 0.000, C 0.000 }
gfCNCPoint1[26036] = {X 575.3370, Y 4.9295, Z -2.1667, A 0.000, B 0.000, C 0.000 }
gfCNCPoint1[26037] = {X 575.3376, Y 5.0000, Z -2.1667, A 0.000, B 0.000, C 0.000 }
gfCNCPoint1[26038] = {X 575.3372, Y 5.9910, Z -2.1667, A 0.000, B 0.000, C 0.000 }
gfCNCPoint1[26039] = {X 575.2576, Y 6.7691, Z -2.1667, A 0.000, B 0.000, C 0.000 }
gfCNCPoint1[26040] = {X 575.0415, Y 7.5209, Z -2.1667, A 0.000, B 0.000, C 0.000 }
gfCNCPoint1[26041] = {X 574.6956, Y 8.2225, Z -2.1667, A 0.000, B 0.000, C 0.000 }
gfCNCPoint1[26042] = {X 575.2866, Y 9.6579, Z -2.1667, A 0.000, B 0.000, C 0.000 }
gfCNCPoint1[26043] = {X 578.9730, Y 18.7113, Z -2.1667, A 0.000, B 0.000, C 0.000 }
gfCNCPoint1[26044] = {X 580.9325, Y 23.5234, Z -2.1667, A 0.000, B 0.000, C 0.000 }
gfCNCPoint1[26045] = {X 581.1912, Y 24.1588, Z -2.1667, A 0.000, B 0.000, C 0.000 }
gfCNCPoint1[26046] = {X 587.7572, Y 8.1004, Z -2.1667, A 0.000, B 0.000, C 0.000 }
gfCNCPoint1[26047] = {X 587.4435, Y 7.4146, Z -2.1667, A 0.000, B 0.000, C 0.000 }
gfCNCPoint1[26048] = {X 587.2516, Y 6.6853, Z -2.1667, A 0.000, B 0.000, C 0.000 }
gfCNCPoint1[26049] = {X 587.1870, Y 5.9339, Z -2.1667, A 0.000, B 0.000, C 0.000 }
gfCNCPoint1[26050] = {X 587.1870, Y 5.0000, Z -2.1667, A 0.000, B 0.000, C 0.000 }
gfCNCPoint1[26051] = {X 587.2780, Y 4.1097, Z -2.1667, A 0.000, B 0.000, C 0.000 }
gfCNCPoint1[26052] = {X 587.5472, Y 3.2562, Z -2.1667, A 0.000, B 0.000, C 0.000 }
gfCNCPoint1[26053] = {X 588.0581, Y 2.3718, Z -2.1667, A 0.000, B 0.000, C 0.000 }
gfCNCPoint1[26054] = {X 588.7592, Y 1.6290, Z -2.1667, A 0.000, B 0.000, C 0.000 }
gfCNCPoint1[26055] = {X 589.6126, Y 1.0678, Z -2.1667, A 0.000, B 0.000, C 0.000 }
gfCNCPoint1[26056] = {X 590.5725, Y 0.7186, Z -2.1667, A 0.000, B 0.000, C 0.000 }
gfCNCPoint1[26057] = {X 591.5870, Y 0.6000, Z -2.1667, A 0.000, B 0.000, C 0.000 }
gfCNCPoint1[26058] = {X 600.0000, Y 0.6000, Z -2.1667, A 0.000, B 0.000, C 0.000 }
gfCNCPoint1[26059] = {X 600.8720, Y 0.6873, Z -2.1667, A 0.000, B 0.000, C 0.000 }
gfCNCPoint1[26060] = {X 601.7094, Y 0.9456, Z -2.1667, A 0.000, B 0.000, C 0.000 }
gfCNCPoint1[26061] = {X 602.4789, Y 1.3648, Z -2.1667, A 0.000, B 0.000, C 0.000 }
gfCNCPoint1[26062] = {X 603.1502, Y 1.9281, Z -2.1667, A 0.000, B 0.000, C 0.000 }
gfCNCPoint1[26063] = {X 603.6965, Y 2.6134, Z -2.1667, A 0.000, B 0.000, C 0.000 }
gfCNCPoint1[26064] = {X 603.6965, Y 1.8140, Z -2.1667, A 0.000, B 0.000, C 0.000 }
gfCNCPoint1[26065] = {X 602.9512, Y 1.1135, Z -2.1667, A 0.000, B 0.000, C 0.000 }
gfCNCPoint1[26066] = {X 602.0762, Y 0.5837, Z -2.1667, A 0.000, B 0.000, C 0.000 }
gfCNCPoint1[26067] = {X 601.1100, Y 0.2479, Z -2.1667, A 0.000, B 0.000, C 0.000 }
gfCNCPoint1[26068] = {X 600.0950, Y 0.1209, Z -2.1667, A 0.000, B 0.000, C 0.000 }
gfCNCPoint1[26069] = {X 600.0948, Y -0.0187, Z -2.1667, A 0.000, B 0.000, C 0.000 }
gfCNCPoint1[26070] = {X 600.0671, Y -0.0697, Z -2.1667, A 0.000, B 0.000, C 0.000 }
gfCNCPoint1[26071] = {X 600.0148, Y -0.0949, Z -2.1667, A 0.000, B 0.000, C 0.000 }
gfCNCPoint1[26072] = {X 351.5626, Y -0.0949, Z -2.1667, A 0.000, B 0.000, C 0.000 }
gfCNCPoint1[26073] = {X 351.4048, Y -0.1241, Z -2.1667, A 0.000, B 0.000, C 0.000 }
gfCNCPoint1[26074] = {X 348.9098, Y -0.4704, Z -2.1667, A 0.000, B 0.000, C 0.000 }
gfCNCPoint1[26075] = {X 346.3934, Y -0.5812, Z -2.1667, A 0.000, B 0.000, C 0.000 }
gfCNCPoint1[26076] = {X 343.8777, Y -0.4557, Z -2.1667, A 0.000, B 0.000, C 0.000 }
gfCNCPoint1[26077] = {X 341.3848, Y -0.0949, Z -2.1667, A 0.000, B 0.000, C 0.000 }
gfCNCPoint1[26078] = {X -0.0148, Y -0.0949, Z -2.1667, A 0.000, B 0.000, C 0.000 }
gfCNCPoint1[26079] = {X -0.0671, Y -0.0697, Z -2.1667, A 0.000, B 0.000, C 0.000 }
gfCNCPoint1[26080] = {X -0.0948, Y -0.0187, Z -2.1667, A 0.000, B 0.000, C 0.000 }
gfCNCPoint1[26081] = {X -0.0965, Y 0.8567, Z -2.1667, A 0.000, B 0.000, C 0.000 }
gfCNCPoint1[26082] = {X -0.0965, Y 8.7890, Z -2.1667, A 0.000, B 0.000, C 0.000 }
gfCNCPoint1[26083] = {X -0.7633, Y 8.9979, Z -2.1667, A 0.000, B 0.000, C 0.000 }
gfCNCPoint1[26084] = {X -1.3935, Y 9.2998, Z -2.1667, A 0.000, B 0.000, C 0.000 }
gfCNCPoint1[26085] = {X -1.9904, Y 9.6404, Z -2.1667, A 0.000, B 0.000, C 0.000 }
gfCNCPoint1[26086] = {X -2.6454, Y 10.0884, Z -2.1667, A 0.000, B 0.000, C 0.000 }
gfCNCPoint1[26087] = {X -3.2192, Y 10.6366, Z -2.1667, A 0.000, B 0.000, C 0.000 }
gfCNCPoint1[26088] = {X -3.6965, Y 11.2705, Z -2.1667, A 0.000, B 0.000, C 0.000 }
gfCNCPoint1[26089] = {X -3.6965, Y 12.3460, Z -2.1667, A 0.000, B 0.000, C 0.000 }
gfCNCPoint1[26090] = {X -3.2331, Y 11.4383, Z -2.1667, A 0.000, B 0.000, C 0.000 }
gfCNCPoint1[26091] = {X -2.5734, Y 10.6615, Z -2.1667, A 0.000, B 0.000, C 0.000 }
gfCNCPoint1[26092] = {X -1.7526, Y 10.0573, Z -2.1667, A 0.000, B 0.000, C 0.000 }
gfCNCPoint1[26093] = {X -1.0994, Y 9.6852, Z -2.1667, A 0.000, B 0.000, C 0.000 }
gfCNCPoint1[26094] = {X -0.1608, Y 9.3012, Z -2.1667, A 0.000, B 0.000, C 0.000 }
gfCNCPoint1[26095] = {X 0.8409, Y 9.1423, Z -2.1667, A 0.000, B 0.000, C 0.000 }
gfCNCPoint1[26096] = {X 1.8522, Y 9.2169, Z -2.1667, A 0.000, B 0.000, C 0.000 }
gfCNCPoint1[26097] = {X 2.2371, Y 9.3087, Z -2.1667, A 0.000, B 0.000, C 0.000 }
gfCNCPoint1[26098] = {X 2.6122, Y 9.4347, Z -2.1667, A 0.000, B 0.000, C 0.000 }
gfCNCPoint1[26099] = {X 3.3800, Y 9.0791, Z -2.1667, A 0.000, B 0.000, C 0.000 }
gfCNCPoint1[26100] = {X 4.1677, Y 8.7700, Z -2.1667, A 0.000, B 0.000, C 0.000 }
gfCNCPoint1[26101] = {X 6.0852, Y 8.0992, Z -2.1667, A 0.000, B 0.000, C 0.000 }
gfCNCPoint1[26102] = {X 8.0533, Y 7.5962, Z -2.1667, A 0.000, B 0.000, C 0.000 }
gfCNCPoint1[26103] = {X 10.0575, Y 7.2646, Z -2.1667, A 0.000, B 0.000, C 0.000 }
gfCNCPoint1[26104] = {X 12.0828, Y 7.1071, Z -2.1667, A 0.000, B 0.000, C 0.000 }
gfCNCPoint1[26105] = {X 14.1141, Y 7.1247, Z -2.1667, A 0.000, B 0.000, C 0.000 }
gfCNCPoint1[26106] = {X 16.1363, Y 7.3173, Z -2.1667, A 0.000, B 0.000, C 0.000 }
gfCNCPoint1[26107] = {X 16.5412, Y 7.3732, Z -2.1667, A 0.000, B 0.000, C 0.000 }
gfCNCPoint1[26108] = {X 17.5022, Y 7.5474, Z -2.1667, A 0.000, B 0.000, C 0.000 }
gfCNCPoint1[26109] = {X 18.4521, Y 7.7747, Z -2.1667, A 0.000, B 0.000, C 0.000 }
gfCNCPoint1[26110] = {X 20.1054, Y 8.3086, Z -2.1667, A 0.000, B 0.000, C 0.000 }
gfCNCPoint1[26111] = {X 21.6977, Y 9.0035, Z -2.1667, A 0.000, B 0.000, C 0.000 }
gfCNCPoint1[26112] = {X 23.2134, Y 9.8524, Z -2.1667, A 0.000, B 0.000, C 0.000 }
gfCNCPoint1[26113] = {X 24.6378, Y 10.8472, Z -2.1667, A 0.000, B 0.000, C 0.000 }
gfCNCPoint1[26114] = {X 25.7295, Y 11.8028, Z -2.1667, A 0.000, B 0.000, C 0.000 }
gfCNCPoint1[26115] = {X 26.7088, Y 12.8732, Z -2.1667, A 0.000, B 0.000, C 0.000 }
gfCNCPoint1[26116] = {X 27.5637, Y 14.0454, Z -2.1667, A 0.000, B 0.000, C 0.000 }
gfCNCPoint1[26117] = {X 28.2837, Y 15.3050, Z -2.1667, A 0.000, B 0.000, C 0.000 }
gfCNCPoint1[26118] = {X 28.8600, Y 16.6365, Z -2.1667, A 0.000, B 0.000, C 0.000 }
gfCNCPoint1[26119] = {X 29.3375, Y 18.3009, Z -2.1667, A 0.000, B 0.000, C 0.000 }
gfCNCPoint1[26120] = {X 29.6207, Y 20.0092, Z -2.1667, A 0.000, B 0.000, C 0.000 }
gfCNCPoint1[26121] = {X 29.7060, Y 21.7387, Z -2.1667, A 0.000, B 0.000, C 0.000 }
gfCNCPoint1[26122] = {X 29.5920, Y 23.4665, Z -2.1667, A 0.000, B 0.000, C 0.000 }
gfCNCPoint1[26123] = {X 29.2804, Y 25.1698, Z -2.1667, A 0.000, B 0.000, C 0.000 }
gfCNCPoint1[26124] = {X 28.7893, Y 26.7454, Z -2.1667, A 0.000, B 0.000, C 0.000 }
gfCNCPoint1[26125] = {X 28.0826, Y 28.2369, Z -2.1667, A 0.000, B 0.000, C 0.000 }
gfCNCPoint1[26126] = {X 27.1742, Y 29.6148, Z -2.1667, A 0.000, B 0.000, C 0.000 }
gfCNCPoint1[26127] = {X 26.3572, Y 30.5720, Z -2.1667, A 0.000, B 0.000, C 0.000 }
gfCNCPoint1[26128] = {X 25.4426, Y 31.4365, Z -2.1667, A 0.000, B 0.000, C 0.000 }
gfCNCPoint1[26129] = {X 25.6932, Y 31.5321, Z -2.1667, A 0.000, B 0.000, C 0.000 }
gfCNCPoint1[26130] = {X 25.9375, Y 31.6428, Z -2.1667, A 0.000, B 0.000, C 0.000 }
gfCNCPoint1[26131] = {X 26.6183, Y 32.0569, Z -2.1667, A 0.000, B 0.000, C 0.000 }
gfCNCPoint1[26132] = {X 27.2131, Y 32.5871, Z -2.1667, A 0.000, B 0.000, C 0.000 }
gfCNCPoint1[26133] = {X 27.2505, Y 32.6275, Z -2.1667, A 0.000, B 0.000, C 0.000 }
gfCNCPoint1[26134] = {X 27.2874, Y 32.6685, Z -2.1667, A 0.000, B 0.000, C 0.000 }
gfCNCPoint1[26135] = {X 27.6590, Y 33.1492, Z -2.1667, A 0.000, B 0.000, C 0.000 }
gfCNCPoint1[26136] = {X 27.9609, Y 33.6766, Z -2.1667, A 0.000, B 0.000, C 0.000 }
gfCNCPoint1[26137] = {X 30.9820, Y 39.9182, Z -2.1667, A 0.000, B 0.000, C 0.000 }
gfCNCPoint1[26138] = {X 31.3085, Y 40.8441, Z -2.1667, A 0.000, B 0.000, C 0.000 }
gfCNCPoint1[26139] = {X 31.4215, Y 41.8194, Z -2.1667, A 0.000, B 0.000, C 0.000 }
gfCNCPoint1[26140] = {X 31.3155, Y 42.7955, Z -2.1667, A 0.000, B 0.000, C 0.000 }
gfCNCPoint1[26141] = {X 30.9956, Y 43.7238, Z -2.1667, A 0.000, B 0.000, C 0.000 }
gfCNCPoint1[26142] = {X 30.4779, Y 44.5580, Z -2.1667, A 0.000, B 0.000, C 0.000 }
gfCNCPoint1[26143] = {X 29.7880, Y 45.2567, Z -2.1667, A 0.000, B 0.000, C 0.000 }
gfCNCPoint1[26144] = {X 29.2516, Y 45.6904, Z -2.1667, A 0.000, B 0.000, C 0.000 }
gfCNCPoint1[26145] = {X 28.5400, Y 46.1588, Z -2.1667, A 0.000, B 0.000, C 0.000 }
gfCNCPoint1[26146] = {X 27.7517, Y 46.4818, Z -2.1667, A 0.000, B 0.000, C 0.000 }
gfCNCPoint1[26147] = {X 26.9160, Y 46.6475, Z -2.1667, A 0.000, B 0.000, C 0.000 }
gfCNCPoint1[26148] = {X 26.0641, Y 46.6498, Z -2.1667, A 0.000, B 0.000, C 0.000 }
gfCNCPoint1[26149] = {X 25.2276, Y 46.4885, Z -2.1667, A 0.000, B 0.000, C 0.000 }
gfCNCPoint1[26150] = {X 23.2128, Y 47.5420, Z -2.1667, A 0.000, B 0.000, C 0.000 }
gfCNCPoint1[26151] = {X 21.1207, Y 48.4320, Z -2.1667, A 0.000, B 0.000, C 0.000 }
gfCNCPoint1[26152] = {X 18.9645, Y 49.1531, Z -2.1667, A 0.000, B 0.000, C 0.000 }
gfCNCPoint1[26153] = {X 17.0292, Y 49.6389, Z -2.1667, A 0.000, B 0.000, C 0.000 }
gfCNCPoint1[26154] = {X 15.0588, Y 49.9531, Z -2.1667, A 0.000, B 0.000, C 0.000 }
gfCNCPoint1[26155] = {X 13.0683, Y 50.0930, Z -2.1667, A 0.000, B 0.000, C 0.000 }
gfCNCPoint1[26156] = {X 11.0733, Y 50.0577, Z -2.1667, A 0.000, B 0.000, C 0.000 }
gfCNCPoint1[26157] = {X 9.0890, Y 49.8475, Z -2.1667, A 0.000, B 0.000, C 0.000 }
gfCNCPoint1[26158] = {X 8.3983, Y 49.7289, Z -2.1667, A 0.000, B 0.000, C 0.000 }
gfCNCPoint1[26159] = {X 8.2281, Y 49.7011, Z -2.1667, A 0.000, B 0.000, C 0.000 }
gfCNCPoint1[26160] = {X 6.5699, Y 49.3108, Z -2.1667, A 0.000, B 0.000, C 0.000 }
gfCNCPoint1[26161] = {X 4.9584, Y 48.7584, Z -2.1667, A 0.000, B 0.000, C 0.000 }
gfCNCPoint1[26162] = {X 3.4095, Y 48.0492, Z -2.1667, A 0.000, B 0.000, C 0.000 }
gfCNCPoint1[26163] = {X 2.3354, Y 47.4416, Z -2.1667, A 0.000, B 0.000, C 0.000 }
gfCNCPoint1[26164] = {X 1.3076, Y 46.7585, Z -2.1667, A 0.000, B 0.000, C 0.000 }
gfCNCPoint1[26165] = {X -0.0255, Y 45.6852, Z -2.1667, A 0.000, B 0.000, C 0.000 }
gfCNCPoint1[26166] = {X -1.2104, Y 44.4502, Z -2.1667, A 0.000, B 0.000, C 0.000 }
gfCNCPoint1[26167] = {X -2.2279, Y 43.0740, Z -2.1667, A 0.000, B 0.000, C 0.000 }
gfCNCPoint1[26168] = {X -3.0611, Y 41.5790, Z -2.1667, A 0.000, B 0.000, C 0.000 }
gfCNCPoint1[26169] = {X -3.6965, Y 39.9898, Z -2.1667, A 0.000, B 0.000, C 0.000 }
gfCNCPoint1[26170] = {X -3.6965, Y 41.3412, Z -2.1667, A 0.000, B 0.000, C 0.000 }
gfCNCPoint1[26171] = {X -3.0078, Y 42.7151, Z -2.1667, A 0.000, B 0.000, C 0.000 }
gfCNCPoint1[26172] = {X -2.1710, Y 44.0041, Z -2.1667, A 0.000, B 0.000, C 0.000 }
gfCNCPoint1[26173] = {X -1.1966, Y 45.1925, Z -2.1667, A 0.000, B 0.000, C 0.000 }
gfCNCPoint1[26174] = {X -0.0965, Y 46.2656, Z -2.1667, A 0.000, B 0.000, C 0.000 }
gfCNCPoint1[26175] = {X -0.0965, Y 99.1433, Z -2.1667, A 0.000, B 0.000, C 0.000 }
gfCNCPoint1[26176] = {X -0.0948, Y 100.0187, Z -2.1667, A 0.000, B 0.000, C 0.000 }
gfCNCPoint1[26177] = {X -0.0671, Y 100.0697, Z -2.1667, A 0.000, B 0.000, C 0.000 }
gfCNCPoint1[26178] = {X -0.0148, Y 100.0949, Z -2.1667, A 0.000, B 0.000, C 0.000 }
gfCNCPoint1[26179] = {X 120.5925, Y 100.0949, Z -2.1667, A 0.000, B 0.000, C 0.000 }
gfCNCPoint1[26180] = {X 121.0613, Y 100.8811, Z -2.1667, A 0.000, B 0.000, C 0.000 }
gfCNCPoint1[26181] = {X 121.6686, Y 101.5660, Z -2.1667, A 0.000, B 0.000, C 0.000 }
gfCNCPoint1[26182] = {X 122.3932, Y 102.1254, Z -2.1667, A 0.000, B 0.000, C 0.000 }
gfCNCPoint1[26183] = {X 123.2094, Y 102.5396, Z -2.1667, A 0.000, B 0.000, C 0.000 }
gfCNCPoint1[26184] = {X 124.0887, Y 102.7942, Z -2.1667, A 0.000, B 0.000, C 0.000 }
gfCNCPoint1[26185] = {X 125.0000, Y 102.8800, Z -2.1667, A 0.000, B 0.000, C 0.000 }
gfCNCPoint1[26186] = {X 143.7791, Y 102.8800, Z -2.1667, A 0.000, B 0.000, C 0.000 }
gfCNCPoint1[26187] = {X 144.6904, Y 102.7942, Z -2.1667, A 0.000, B 0.000, C 0.000 }
gfCNCPoint1[26188] = {X 145.5697, Y 102.5396, Z -2.1667, A 0.000, B 0.000, C 0.000 }
gfCNCPoint1[26189] = {X 146.3859, Y 102.1254, Z -2.1667, A 0.000, B 0.000, C 0.000 }
gfCNCPoint1[26190] = {X 147.1105, Y 101.5660, Z -2.1667, A 0.000, B 0.000, C 0.000 }
gfCNCPoint1[26191] = {X 147.7178, Y 100.8811, Z -2.1667, A 0.000, B 0.000, C 0.000 }
gfCNCPoint1[26192] = {X 148.1866, Y 100.0949, Z -2.1667, A 0.000, B 0.000, C 0.000 }
gfCNCPoint1[26193] = {X 150.8372, Y 100.0949, Z -2.1667, A 0.000, B 0.000, C 0.000 }
gfCNCPoint1[26194] = {X 150.8372, Y 95.2949, Z -2.1667, A 0.000, B 0.000, C 0.000 }
gfCNCPoint1[26195] = {X 187.9257, Y 95.2949, Z -2.1667, A 0.000, B 0.000, C 0.000 }
gfCNCPoint1[26196] = {X 187.9777, Y 95.0989, Z -2.1667, A 0.000, B 0.000, C 0.000 }
gfCNCPoint1[26197] = {X 188.0352, Y 94.9045, Z -2.1667, A 0.000, B 0.000, C 0.000 }
gfCNCPoint1[26198] = {X 187.2619, Y 94.0602, Z -2.1667, A 0.000, B 0.000, C 0.000 }
gfCNCPoint1[26199] = {X 151.4055, Y 94.0602, Z -2.1667, A 0.000, B 0.000, C 0.000 }
gfCNCPoint1[26200] = {X 150.7053, Y 94.8360, Z -2.1667, A 0.000, B 0.000, C 0.000 }
gfCNCPoint1[26201] = {X 150.7750, Y 95.0644, Z -2.1667, A 0.000, B 0.000, C 0.000 }
gfCNCPoint1[26202] = {X 150.8372, Y 95.2949, Z -2.1667, A 0.000, B 0.000, C 0.000 }
gfCNCPoint1[26203] = {X 150.8372, Y 97.6949, Z -2.1667, A 0.000, B 0.000, C 0.000 }
gfCNCPoint1[26204] = {X 190.1070, Y 97.6949, Z -2.1667, A 0.000, B 0.000, C 0.000 }
gfCNCPoint1[26205] = {X 190.1070, Y 97.0659, Z -2.1667, A 0.000, B 0.000, C 0.000 }
gfCNCPoint1[26206] = {X 190.1938, Y 96.1495, Z -2.1667, A 0.000, B 0.000, C 0.000 }
gfCNCPoint1[26207] = {X 190.4511, Y 95.2657, Z -2.1667, A 0.000, B 0.000, C 0.000 }
gfCNCPoint1[26208] = {X 190.8699, Y 94.4460, Z -2.1667, A 0.000, B 0.000, C 0.000 }
gfCNCPoint1[26209] = {X 188.3182, Y 91.6602, Z -2.1667, A 0.000, B 0.000, C 0.000 }
gfCNCPoint1[26210] = {X 150.3387, Y 91.6602, Z -2.1667, A 0.000, B 0.000, C 0.000 }
gfCNCPoint1[26211] = {X 147.8633, Y 94.4027, Z -2.1667, A 0.000, B 0.000, C 0.000 }
gfCNCPoint1[26212] = {X 148.2974, Y 95.2329, Z -2.1667, A 0.000, B 0.000, C 0.000 }
gfCNCPoint1[26213] = {X 148.5659, Y 96.1303, Z -2.1667, A 0.000, B 0.000, C 0.000 }
gfCNCPoint1[26214] = {X 148.6591, Y 97.0625, Z -2.1667, A 0.000, B 0.000, C 0.000 }
gfCNCPoint1[26215] = {X 148.6591, Y 97.6949, Z -2.1667, A 0.000, B 0.000, C 0.000 }
gfCNCPoint1[26216] = {X 150.8372, Y 97.6949, Z -2.1667, A 0.000, B 0.000, C 0.000 }
gfCNCPoint1[26217] = {X 150.8372, Y 100.0949, Z -2.1667, A 0.000, B 0.000, C 0.000 }
gfCNCPoint1[26218] = {X 190.5795, Y 100.0949, Z -2.1667, A 0.000, B 0.000, C 0.000 }
gfCNCPoint1[26219] = {X 191.0483, Y 100.8811, Z -2.1667, A 0.000, B 0.000, C 0.000 }
gfCNCPoint1[26220] = {X 191.6556, Y 101.5660, Z -2.1667, A 0.000, B 0.000, C 0.000 }
gfCNCPoint1[26221] = {X 192.3801, Y 102.1254, Z -2.1667, A 0.000, B 0.000, C 0.000 }
gfCNCPoint1[26222] = {X 193.1964, Y 102.5396, Z -2.1667, A 0.000, B 0.000, C 0.000 }
gfCNCPoint1[26223] = {X 194.0756, Y 102.7942, Z -2.1667, A 0.000, B 0.000, C 0.000 }
gfCNCPoint1[26224] = {X 194.9870, Y 102.8800, Z -2.1667, A 0.000, B 0.000, C 0.000 }
gfCNCPoint1[26225] = {X 212.6141, Y 102.8800, Z -2.1667, A 0.000, B 0.000, C 0.000 }
gfCNCPoint1[26226] = {X 213.0066, Y 102.8642, Z -2.1667, A 0.000, B 0.000, C 0.000 }
gfCNCPoint1[26227] = {X 213.3966, Y 102.8169, Z -2.1667, A 0.000, B 0.000, C 0.000 }
gfCNCPoint1[26228] = {X 213.7865, Y 102.8642, Z -2.1667, A 0.000, B 0.000, C 0.000 }
gfCNCPoint1[26229] = {X 214.1790, Y 102.8800, Z -2.1667, A 0.000, B 0.000, C 0.000 }
gfCNCPoint1[26230] = {X 233.4798, Y 102.8800, Z -2.1667, A 0.000, B 0.000, C 0.000 }
gfCNCPoint1[26231] = {X 234.3911, Y 102.7942, Z -2.1667, A 0.000, B 0.000, C 0.000 }
gfCNCPoint1[26232] = {X 235.2704, Y 102.5396, Z -2.1667, A 0.000, B 0.000, C 0.000 }
gfCNCPoint1[26233] = {X 236.0866, Y 102.1254, Z -2.1667, A 0.000, B 0.000, C 0.000 }
gfCNCPoint1[26234] = {X 236.8112, Y 101.5660, Z -2.1667, A 0.000, B 0.000, C 0.000 }
gfCNCPoint1[26235] = {X 237.4185, Y 100.8811, Z -2.1667, A 0.000, B 0.000, C 0.000 }
gfCNCPoint1[26236] = {X 237.8872, Y 100.0949, Z -2.1667, A 0.000, B 0.000, C 0.000 }
gfCNCPoint1[26237] = {X 261.4768, Y 100.0949, Z -2.1667, A 0.000, B 0.000, C 0.000 }
gfCNCPoint1[26238] = {X 261.4768, Y 90.4949, Z -2.1667, A 0.000, B 0.000, C 0.000 }
gfCNCPoint1[26239] = {X 266.0962, Y 90.4949, Z -2.1667, A 0.000, B 0.000, C 0.000 }
gfCNCPoint1[26240] = {X 266.1752, Y 90.3747, Z -2.1667, A 0.000, B 0.000, C 0.000 }
gfCNCPoint1[26241] = {X 266.2556, Y 90.2554, Z -2.1667, A 0.000, B 0.000, C 0.000 }
gfCNCPoint1[26242] = {X 263.5089, Y 89.1787, Z -2.1667, A 0.000, B 0.000, C 0.000 }
gfCNCPoint1[26243] = {X 261.4768, Y 90.4949, Z -2.1667, A 0.000, B 0.000, C 0.000 }
gfCNCPoint1[26244] = {X 261.4768, Y 92.8949, Z -2.1667, A 0.000, B 0.000, C 0.000 }
gfCNCPoint1[26245] = {X 267.4974, Y 92.8949, Z -2.1667, A 0.000, B 0.000, C 0.000 }
gfCNCPoint1[26246] = {X 267.8429, Y 92.2375, Z -2.1667, A 0.000, B 0.000, C 0.000 }
gfCNCPoint1[26247] = {X 268.2378, Y 91.6085, Z -2.1667, A 0.000, B 0.000, C 0.000 }
gfCNCPoint1[26248] = {X 269.1700, Y 90.4463, Z -2.1667, A 0.000, B 0.000, C 0.000 }
gfCNCPoint1[26249] = {X 270.2694, Y 89.4409, Z -2.1667, A 0.000, B 0.000, C 0.000 }
gfCNCPoint1[26250] = {X 270.2694, Y 89.2510, Z -2.1667, A 0.000, B 0.000, C 0.000 }
gfCNCPoint1[26251] = {X 263.2380, Y 86.4947, Z -2.1667, A 0.000, B 0.000, C 0.000 }
gfCNCPoint1[26252] = {X 253.3569, Y 92.8949, Z -2.1667, A 0.000, B 0.000, C 0.000 }
gfCNCPoint1[26253] = {X 261.4768, Y 92.8949, Z -2.1667, A 0.000, B 0.000, C 0.000 }
gfCNCPoint1[26254] = {X 261.4768, Y 95.2949, Z -2.1667, A 0.000, B 0.000, C 0.000 }
gfCNCPoint1[26255] = {X 269.1714, Y 95.2949, Z -2.1667, A 0.000, B 0.000, C 0.000 }
gfCNCPoint1[26256] = {X 269.5516, Y 94.1744, Z -2.1667, A 0.000, B 0.000, C 0.000 }
gfCNCPoint1[26257] = {X 270.1083, Y 93.1302, Z -2.1667, A 0.000, B 0.000, C 0.000 }
gfCNCPoint1[26258] = {X 270.8267, Y 92.1901, Z -2.1667, A 0.000, B 0.000, C 0.000 }
gfCNCPoint1[26259] = {X 271.6880, Y 91.3787, Z -2.1667, A 0.000, B 0.000, C 0.000 }
gfCNCPoint1[26260] = {X 272.6694, Y 90.7176, Z -2.1667, A 0.000, B 0.000, C 0.000 }
gfCNCPoint1[26261] = {X 272.6694, Y 87.6139, Z -2.1667, A 0.000, B 0.000, C 0.000 }
gfCNCPoint1[26262] = {X 262.9671, Y 83.8107, Z -2.1667, A 0.000, B 0.000, C 0.000 }
gfCNCPoint1[26263] = {X 245.2369, Y 95.2949, Z -2.1667, A 0.000, B 0.000, C 0.000 }
gfCNCPoint1[26264] = {X 261.4768, Y 95.2949, Z -2.1667, A 0.000, B 0.000, C 0.000 }
gfCNCPoint1[26265] = {X 261.4768, Y 97.6949, Z -2.1667, A 0.000, B 0.000, C 0.000 }
gfCNCPoint1[26266] = {X 271.3527, Y 97.6949, Z -2.1667, A 0.000, B 0.000, C 0.000 }
gfCNCPoint1[26267] = {X 271.3529, Y 97.0186, Z -2.1667, A 0.000, B 0.000, C 0.000 }
gfCNCPoint1[26268] = {X 271.4810, Y 95.9545, Z -2.1667, A 0.000, B 0.000, C 0.000 }
gfCNCPoint1[26269] = {X 271.8382, Y 94.9440, Z -2.1667, A 0.000, B 0.000, C 0.000 }
gfCNCPoint1[26270] = {X 272.4073, Y 94.0359, Z -2.1667, A 0.000, B 0.000, C 0.000 }
gfCNCPoint1[26271] = {X 273.1610, Y 93.2739, Z -2.1667, A 0.000, B 0.000, C 0.000 }
gfCNCPoint1[26272] = {X 274.0629, Y 92.6949, Z -2.1667, A 0.000, B 0.000, C 0.000 }
gfCNCPoint1[26273] = {X 275.0694, Y 92.3266, Z -2.1667, A 0.000, B 0.000, C 0.000 }
gfCNCPoint1[26274] = {X 275.0694, Y 85.9769, Z -2.1667, A 0.000, B 0.000, C 0.000 }
gfCNCPoint1[26275] = {X 262.6984, Y 81.1275, Z -2.1667, A 0.000, B 0.000, C 0.000 }
gfCNCPoint1[26276] = {X 262.5773, Y 81.2037, Z -2.1667, A 0.000, B 0.000, C 0.000 }
gfCNCPoint1[26277] = {X 238.3584, Y 96.8908, Z -2.1667, A 0.000, B 0.000, C 0.000 }
gfCNCPoint1[26278] = {X 238.3598, Y 97.0659, Z -2.1667, A 0.000, B 0.000, C 0.000 }
gfCNCPoint1[26279] = {X 238.3598, Y 97.6949, Z -2.1667, A 0.000, B 0.000, C 0.000 }
gfCNCPoint1[26280] = {X 261.4768, Y 97.6949, Z -2.1667, A 0.000, B 0.000, C 0.000 }
gfCNCPoint1[26281] = {X 261.4768, Y 100.0949, Z -2.1667, A 0.000, B 0.000, C 0.000 }
gfCNCPoint1[26282] = {X 271.8252, Y 100.0949, Z -2.1667, A 0.000, B 0.000, C 0.000 }
gfCNCPoint1[26283] = {X 272.2940, Y 100.8811, Z -2.1667, A 0.000, B 0.000, C 0.000 }
gfCNCPoint1[26284] = {X 272.9013, Y 101.5660, Z -2.1667, A 0.000, B 0.000, C 0.000 }
gfCNCPoint1[26285] = {X 273.6259, Y 102.1254, Z -2.1667, A 0.000, B 0.000, C 0.000 }
gfCNCPoint1[26286] = {X 274.4421, Y 102.5396, Z -2.1667, A 0.000, B 0.000, C 0.000 }
gfCNCPoint1[26287] = {X 275.3214, Y 102.7942, Z -2.1667, A 0.000, B 0.000, C 0.000 }
gfCNCPoint1[26288] = {X 276.2327, Y 102.8800, Z -2.1667, A 0.000, B 0.000, C 0.000 }
gfCNCPoint1[26289] = {X 292.7731, Y 102.8800, Z -2.1667, A 0.000, B 0.000, C 0.000 }
gfCNCPoint1[26290] = {X 293.6844, Y 102.7942, Z -2.1667, A 0.000, B 0.000, C 0.000 }
gfCNCPoint1[26291] = {X 294.5637, Y 102.5396, Z -2.1667, A 0.000, B 0.000, C 0.000 }
gfCNCPoint1[26292] = {X 295.3799, Y 102.1254, Z -2.1667, A 0.000, B 0.000, C 0.000 }
gfCNCPoint1[26293] = {X 296.1045, Y 101.5660, Z -2.1667, A 0.000, B 0.000, C 0.000 }
gfCNCPoint1[26294] = {X 296.7118, Y 100.8811, Z -2.1667, A 0.000, B 0.000, C 0.000 }
gfCNCPoint1[26295] = {X 297.1805, Y 100.0949, Z -2.1667, A 0.000, B 0.000, C 0.000 }
gfCNCPoint1[26296] = {X 319.1366, Y 100.0949, Z -2.1667, A 0.000, B 0.000, C 0.000 }
gfCNCPoint1[26297] = {X 321.4385, Y 100.8673, Z -2.1667, A 0.000, B 0.000, C 0.000 }
gfCNCPoint1[26298] = {X 323.7829, Y 101.4989, Z -2.1667, A 0.000, B 0.000, C 0.000 }
gfCNCPoint1[26299] = {X 326.1612, Y 101.9874, Z -2.1667, A 0.000, B 0.000, C 0.000 }
gfCNCPoint1[26300] = {X 329.6396, Y 102.5409, Z -2.1667, A 0.000, B 0.000, C 0.000 }
gfCNCPoint1[26301] = {X 333.1371, Y 102.9564, Z -2.1667, A 0.000, B 0.000, C 0.000 }
gfCNCPoint1[26302] = {X 336.6483, Y 103.2331, Z -2.1667, A 0.000, B 0.000, C 0.000 }
gfCNCPoint1[26303] = {X 342.8092, Y 103.5151, Z -2.1667, A 0.000, B 0.000, C 0.000 }
gfCNCPoint1[26304] = {X 348.9761, Y 103.5917, Z -2.1667, A 0.000, B 0.000, C 0.000 }
gfCNCPoint1[26305] = {X 355.1421, Y 103.4628, Z -2.1667, A 0.000, B 0.000, C 0.000 }
gfCNCPoint1[26306] = {X 361.3005, Y 103.1286, Z -2.1667, A 0.000, B 0.000, C 0.000 }
gfCNCPoint1[26307] = {X 365.1928, Y 102.7581, Z -2.1667, A 0.000, B 0.000, C 0.000 }
gfCNCPoint1[26308] = {X 369.0628, Y 102.2007, Z -2.1667, A 0.000, B 0.000, C 0.000 }
gfCNCPoint1[26309] = {X 372.9015, Y 101.4580, Z -2.1667, A 0.000, B 0.000, C 0.000 }
gfCNCPoint1[26310] = {X 375.2293, Y 100.8561, Z -2.1667, A 0.000, B 0.000, C 0.000 }
gfCNCPoint1[26311] = {X 377.5099, Y 100.0949, Z -2.1667, A 0.000, B 0.000, C 0.000 }
gfCNCPoint1[26312] = {X 391.9985, Y 100.0949, Z -2.1667, A 0.000, B 0.000, C 0.000 }
gfCNCPoint1[26313] = {X 392.4672, Y 100.8811, Z -2.1667, A 0.000, B 0.000, C 0.000 }
gfCNCPoint1[26314] = {X 393.0746, Y 101.5660, Z -2.1667, A 0.000, B 0.000, C 0.000 }
gfCNCPoint1[26315] = {X 393.7991, Y 102.1254, Z -2.1667, A 0.000, B 0.000, C 0.000 }
gfCNCPoint1[26316] = {X 394.6154, Y 102.5396, Z -2.1667, A 0.000, B 0.000, C 0.000 }
gfCNCPoint1[26317] = {X 395.4946, Y 102.7942, Z -2.1667, A 0.000, B 0.000, C 0.000 }
gfCNCPoint1[26318] = {X 396.4059, Y 102.8800, Z -2.1667, A 0.000, B 0.000, C 0.000 }
gfCNCPoint1[26319] = {X 415.7067, Y 102.8800, Z -2.1667, A 0.000, B 0.000, C 0.000 }
gfCNCPoint1[26320] = {X 416.6180, Y 102.7942, Z -2.1667, A 0.000, B 0.000, C 0.000 }
gfCNCPoint1[26321] = {X 417.4973, Y 102.5396, Z -2.1667, A 0.000, B 0.000, C 0.000 }
gfCNCPoint1[26322] = {X 418.3135, Y 102.1254, Z -2.1667, A 0.000, B 0.000, C 0.000 }
gfCNCPoint1[26323] = {X 419.0381, Y 101.5660, Z -2.1667, A 0.000, B 0.000, C 0.000 }
gfCNCPoint1[26324] = {X 419.6454, Y 100.8811, Z -2.1667, A 0.000, B 0.000, C 0.000 }
gfCNCPoint1[26325] = {X 420.1142, Y 100.0949, Z -2.1667, A 0.000, B 0.000, C 0.000 }
gfCNCPoint1[26326] = {X 443.7015, Y 100.0949, Z -2.1667, A 0.000, B 0.000, C 0.000 }
gfCNCPoint1[26327] = {X 443.7015, Y 90.4949, Z -2.1667, A 0.000, B 0.000, C 0.000 }
gfCNCPoint1[26328] = {X 448.3231, Y 90.4949, Z -2.1667, A 0.000, B 0.000, C 0.000 }
gfCNCPoint1[26329] = {X 448.4021, Y 90.3747, Z -2.1667, A 0.000, B 0.000, C 0.000 }
gfCNCPoint1[26330] = {X 448.4825, Y 90.2554, Z -2.1667, A 0.000, B 0.000, C 0.000 }
gfCNCPoint1[26331] = {X 445.7343, Y 89.1781, Z -2.1667, A 0.000, B 0.000, C 0.000 }
gfCNCPoint1[26332] = {X 443.7015, Y 90.4949, Z -2.1667, A 0.000, B 0.000, C 0.000 }
gfCNCPoint1[26333] = {X 443.7015, Y 92.8949, Z -2.1667, A 0.000, B 0.000, C 0.000 }
gfCNCPoint1[26334] = {X 449.7243, Y 92.8949, Z -2.1667, A 0.000, B 0.000, C 0.000 }
gfCNCPoint1[26335] = {X 450.0698, Y 92.2375, Z -2.1667, A 0.000, B 0.000, C 0.000 }
gfCNCPoint1[26336] = {X 450.4647, Y 91.6084, Z -2.1667, A 0.000, B 0.000, C 0.000 }
gfCNCPoint1[26337] = {X 451.3969, Y 90.4463, Z -2.1667, A 0.000, B 0.000, C 0.000 }
gfCNCPoint1[26338] = {X 452.4963, Y 89.4409, Z -2.1667, A 0.000, B 0.000, C 0.000 }
gfCNCPoint1[26339] = {X 452.4963, Y 89.2510, Z -2.1667, A 0.000, B 0.000, C 0.000 }
gfCNCPoint1[26340] = {X 445.4633, Y 86.4940, Z -2.1667, A 0.000, B 0.000, C 0.000 }
gfCNCPoint1[26341] = {X 435.5823, Y 92.8949, Z -2.1667, A 0.000, B 0.000, C 0.000 }
gfCNCPoint1[26342] = {X 443.7015, Y 92.8949, Z -2.1667, A 0.000, B 0.000, C 0.000 }
gfCNCPoint1[26343] = {X 443.7015, Y 95.2949, Z -2.1667, A 0.000, B 0.000, C 0.000 }
gfCNCPoint1[26344] = {X 451.3983, Y 95.2949, Z -2.1667, A 0.000, B 0.000, C 0.000 }
gfCNCPoint1[26345] = {X 451.7785, Y 94.1744, Z -2.1667, A 0.000, B 0.000, C 0.000 }
gfCNCPoint1[26346] = {X 452.3352, Y 93.1302, Z -2.1667, A 0.000, B 0.000, C 0.000 }
gfCNCPoint1[26347] = {X 453.0536, Y 92.1901, Z -2.1667, A 0.000, B 0.000, C 0.000 }
gfCNCPoint1[26348] = {X 453.9149, Y 91.3787, Z -2.1667, A 0.000, B 0.000, C 0.000 }
gfCNCPoint1[26349] = {X 454.8963, Y 90.7176, Z -2.1667, A 0.000, B 0.000, C 0.000 }
gfCNCPoint1[26350] = {X 454.8963, Y 87.6139, Z -2.1667, A 0.000, B 0.000, C 0.000 }
gfCNCPoint1[26351] = {X 445.1924, Y 83.8100, Z -2.1667, A 0.000, B 0.000, C 0.000 }
gfCNCPoint1[26352] = {X 427.4632, Y 95.2949, Z -2.1667, A 0.000, B 0.000, C 0.000 }
gfCNCPoint1[26353] = {X 443.7015, Y 95.2949, Z -2.1667, A 0.000, B 0.000, C 0.000 }
gfCNCPoint1[26354] = {X 443.7015, Y 97.6949, Z -2.1667, A 0.000, B 0.000, C 0.000 }
gfCNCPoint1[26355] = {X 453.5796, Y 97.6949, Z -2.1667, A 0.000, B 0.000, C 0.000 }
gfCNCPoint1[26356] = {X 453.5796, Y 97.0659, Z -2.1667, A 0.000, B 0.000, C 0.000 }
gfCNCPoint1[26357] = {X 453.6990, Y 95.9930, Z -2.1667, A 0.000, B 0.000, C 0.000 }
gfCNCPoint1[26358] = {X 454.0514, Y 94.9725, Z -2.1667, A 0.000, B 0.000, C 0.000 }
gfCNCPoint1[26359] = {X 454.6196, Y 94.0545, Z -2.1667, A 0.000, B 0.000, C 0.000 }
gfCNCPoint1[26360] = {X 455.3757, Y 93.2839, Z -2.1667, A 0.000, B 0.000, C 0.000 }
gfCNCPoint1[26361] = {X 456.2827, Y 92.6984, Z -2.1667, A 0.000, B 0.000, C 0.000 }
gfCNCPoint1[26362] = {X 457.2963, Y 92.3266, Z -2.1667, A 0.000, B 0.000, C 0.000 }
gfCNCPoint1[26363] = {X 457.2963, Y 85.9769, Z -2.1667, A 0.000, B 0.000, C 0.000 }
gfCNCPoint1[26364] = {X 444.9214, Y 81.1260, Z -2.1667, A 0.000, B 0.000, C 0.000 }
gfCNCPoint1[26365] = {X 420.5853, Y 96.8909, Z -2.1667, A 0.000, B 0.000, C 0.000 }
gfCNCPoint1[26366] = {X 420.5867, Y 97.0659, Z -2.1667, A 0.000, B 0.000, C 0.000 }
gfCNCPoint1[26367] = {X 420.5867, Y 97.6949, Z -2.1667, A 0.000, B 0.000, C 0.000 }
gfCNCPoint1[26368] = {X 443.7015, Y 97.6949, Z -2.1667, A 0.000, B 0.000, C 0.000 }
gfCNCPoint1[26369] = {X 443.7015, Y 100.0949, Z -2.1667, A 0.000, B 0.000, C 0.000 }
gfCNCPoint1[26370] = {X 454.0521, Y 100.0949, Z -2.1667, A 0.000, B 0.000, C 0.000 }
gfCNCPoint1[26371] = {X 454.5209, Y 100.8811, Z -2.1667, A 0.000, B 0.000, C 0.000 }
gfCNCPoint1[26372] = {X 455.1282, Y 101.5660, Z -2.1667, A 0.000, B 0.000, C 0.000 }
gfCNCPoint1[26373] = {X 455.8528, Y 102.1254, Z -2.1667, A 0.000, B 0.000, C 0.000 }
gfCNCPoint1[26374] = {X 456.6690, Y 102.5396, Z -2.1667, A 0.000, B 0.000, C 0.000 }
gfCNCPoint1[26375] = {X 457.5483, Y 102.7942, Z -2.1667, A 0.000, B 0.000, C 0.000 }
gfCNCPoint1[26376] = {X 458.4596, Y 102.8800, Z -2.1667, A 0.000, B 0.000, C 0.000 }
gfCNCPoint1[26377] = {X 475.0000, Y 102.8800, Z -2.1667, A 0.000, B 0.000, C 0.000 }
gfCNCPoint1[26378] = {X 475.9113, Y 102.7942, Z -2.1667, A 0.000, B 0.000, C 0.000 }
gfCNCPoint1[26379] = {X 476.7906, Y 102.5396, Z -2.1667, A 0.000, B 0.000, C 0.000 }
gfCNCPoint1[26380] = {X 477.6068, Y 102.1254, Z -2.1667, A 0.000, B 0.000, C 0.000 }
gfCNCPoint1[26381] = {X 478.3314, Y 101.5660, Z -2.1667, A 0.000, B 0.000, C 0.000 }
gfCNCPoint1[26382] = {X 478.9387, Y 100.8811, Z -2.1667, A 0.000, B 0.000, C 0.000 }
gfCNCPoint1[26383] = {X 479.4075, Y 100.0949, Z -2.1667, A 0.000, B 0.000, C 0.000 }
gfCNCPoint1[26384] = {X 507.6819, Y 100.0949, Z -2.1667, A 0.000, B 0.000, C 0.000 }
gfCNCPoint1[26385] = {X 507.6819, Y 107.6949, Z -2.1667, A 0.000, B 0.000, C 0.000 }
gfCNCPoint1[26386] = {X 507.6819, Y 107.6949, Z 0.8333, A 0.000, B 0.000, C 0.000 }
gfCNCPoint1[26387] = {X 507.6819, Y 107.6949, Z 11.0000, A 0.000, B 0.000, C 0.000 }
gfCNCPoint1[26388] = {X 108.5557, Y 40.9005, Z 11.0000, A 0.000, B 0.000, C 0.000 }
gfCNCPoint1[26389] = {X 108.5557, Y 40.9005, Z 1.6667, A 0.000, B 0.000, C 0.000 }
gfCNCPoint1[26390] = {X 108.5557, Y 40.9005, Z -2.1667, A 0.000, B 0.000, C 0.000 }
gfCNCPoint1[26391] = {X 108.0646, Y 42.1007, Z -2.1667, A 0.000, B 0.000, C 0.000 }
gfCNCPoint1[26392] = {X 108.0890, Y 42.0581, Z -2.1667, A 0.000, B 0.000, C 0.000 }
gfCNCPoint1[26393] = {X 108.1138, Y 42.0159, Z -2.1667, A 0.000, B 0.000, C 0.000 }
gfCNCPoint1[26394] = {X 108.5422, Y 41.3922, Z -2.1667, A 0.000, B 0.000, C 0.000 }
